(* IEC 61131-3 sources: elnaProjects/ElpcLogic/PomarKc7Changed/build_USO_ecl (part 4) *)

      (*Режим ЭГПА остановлен *)
      EGPA_Stop.top := (algManager.mode = ModeGpa.MODE_STOP);

      (*Автомат ШУ включен *)
      Avt_SHU_vkl.top := IM.SingleSignals.SHU_v_GPA_vkluch.Q;

      (*Все исполнительные механизмы выключены *)
      All_IM_Off.top := (IM.mv.onStatus=_statusDualInput.STATUS_OFF) AND (IM.pns.onStatus=_statusDualInput.STATUS_OFF) AND
                        (IM.nu1.onStatus=_statusDualInput.STATUS_OFF) AND (IM.nu2.onStatus=_statusDualInput.STATUS_OFF) AND
                        (IM.v1_Avom.onStatus=_statusDualInput.STATUS_OFF) AND (IM.v2_Avom.onStatus=_statusDualInput.STATUS_OFF) AND
  		  (IM.v3_Avom.onStatus=_statusDualInput.STATUS_OFF)AND (IM.v4_Avom.onStatus=_statusDualInput.STATUS_OFF) AND
                        (IM.CMN.onStatus=_statusDualInput.STATUS_OFF) AND (IM.TEN_MB.onStatus=_statusDualInput.STATUS_OFF) AND
                        (IM.TEN_kollectora.onStatus=_statusDualInput.STATUS_OFF) AND (IM.KaloriferAVOM.onStatus=_statusDualInput.STATUS_OFF);

      (*Наличие 220 в шу*)
      Nalichie220_SHU_Ai.top :=	(ai.Kontrol_per_220V.interval = _statusAi.normal)	 AND (ai.Kontrol_post_220V.interval = _statusAi.normal);

      (*Блоки питания норм*)
      BP_Norm.top:=
  		(IM.SingleSignals.Nalichie_BP1.Q AND
  		IM.SingleSignals.Nalichie_BP2.Q AND
  		IM.SingleSignals.Nalichie_BP3.Q AND
  		IM.SingleSignals.Nalichie_BP4.Q AND
  		IM.SingleSignals.Nalichie_BP5.Q AND
  		IM.SingleSignals.Nalichie_BP6.Q AND
  		IM.SingleSignals.Nalichie_BP7_BP8.Q AND
  		IM.SingleSignals.Nalichie_BP9_BP10.Q AND

  		IM.SingleSignals.Nalichie_220BEAO.Q AND
  		IM.SingleSignals.Nalichie_per_220_na_vhode.Q AND
  		IM.SingleSignals.Nalichie_post_220_na_vhode.Q AND
  		IM.SingleSignals.Nalichie_BP11.Q AND
  		IM.SingleSignals.Nalichie_BP12.Q);

      (*Напряжение исполнительниых механизмов
      Naprajenie_U_IM.top := IM.NalichieU_CMN.q AND IM.NalichieU_NU1.Q AND IM.Nalichie_CU_MV.Q  AND IM.NalichieU_NU2.Q AND
  						IM.NalichieU_PNS.Q; нет сигналов таких *)

      (* положение тележки мв вкачена *)
      MV_Poloj_RolledON.top:= IM.mv.basketStatus = _basketStats.BASKET_ROLLEDIN;

      (* положение тележки мв выкачена *)
      MV_Poloj_RolledOFF.top:= IM.mv.basketStatus = _basketStats.BASKET_ROLLEDOUT;

      (* нет неисправных аналоговых сигналов *)
      NOTAnalogNS.top :=  NOT analogsNS();

      (* нет аварийных/предупредительных сигнализаций аналоговых сигналов *)
      Net_ASPS_Analogs.top := anyAnalogsPs(); (*Не понял где посмотреть наличие ас аналогов *)

      (* нет сработанных защит *)
      Not_AS.top := NOT anyProtectionSignaling();

      (* готовность возбудителя *)
      Gotov_Vozb.top:= IM.SingleSignals.Vozbud_gotovnost.Q;

      (* реакторный пуск *)
      (*Reactornyi_P.top := IM.SingleSignals.Reaktornii_pusk_perek.Q AND NOT IM.SingleSignals.Chastotny_pusk.Q;*)

      (* частотный пуск *)
     (* Chastotnyi_P.top:=IM.SingleSignals.Chastotny_pusk.Q AND NOT IM.SingleSignals.Reaktornii_pusk_perek.Q;*)

      (* нет перепада давления на кране 1 *)
      dP_kr1.top:= NOT IM.SingleSignals.dp_kran1_Less100.Q (*AND (IM.PerepadDavlenieKran1_CK.status = 1))*);

      (* в автоматическом ли режиме исполнительные механизмы *)
      (*Auto_Rej.top := im.NU1_Automat.Q AND im.PNS_Automat.Q AND im.NU2_Automat.Q;*)

      (* есть наряжение в цепях управления ИМ *)
      CK_IM_Norm.top := nsCepeiUpravlenya();

      (* ручной режим *)
      HAnd_Mode.top:= NOT im.SingleSignals.Rezhim_ruchnogo_regulirovaniya.Q;

      (* импульсный газ *)
      Impuls_Gaz.top:= ai.Pimpuls_gaz.interval=_statusAi.normal;

      ppuDone := BMP_Err.top AND
  	     Level_masla_Norm.top AND
                 T_masla_Norm.top AND
  	     Krans_ready_to_move.top AND
  	     Krans_Poloj.top AND
  	     Net_AO_KC_SHKS04M.top AND
  	     EGPA_Stop.top AND
                 Avt_SHU_vkl.top AND
                 All_IM_Off.top AND
                 Nalichie220_SHU_Ai.top AND
                 BP_Norm.top AND
                 Naprajenie_U_IM.top AND
                 MV_Poloj_RolledON.top AND
                 MV_Poloj_RolledOFF.top AND
                 NOTAnalogNS.top AND
                 Net_ASPS_Analogs.top AND
                 Not_AS.top AND
                 Gotov_Vozb.top AND
                 Reactornyi_P.top AND
                 Chastotnyi_P.top AND
                 dP_kr1.top AND
                 Auto_Rej.top AND
                 CK_IM_Norm.top AND
                 HAnd_Mode.top AND
                 Impuls_Gaz.top;

      puskAllowed:= ppuDone AND Im.mv.basketStatus = _basketStats.BASKET_ROLLEDIN;
      testAllowed:= ppuDone AND Im.mv.basketStatus = _basketStats.BASKET_ROLLEDOUT;

      modeR_Trig(CLK:=puskAllowed);
      modeF_Trig(CLK:=puskAllowed);

      IF modeR_Trig.Q THEN
  	algManager.nMode:= ModeGpa.MODE_READY;
      END_IF;
      IF modeF_Trig.Q THEN
  	algManager.nMode:= ModeGpa.MODE_STOP;
      END_IF;

      IF puskAllowed THEN
          algoritms.Apusk.inCanRun:= TRUE;
          algoritms.SemiAutoPusk.inCanRun:= TRUE;
      ELSE
          algoritms.Apusk.inCanRun:= FALSE;
          algoritms.SemiAutoPusk.inCanRun:= FALSE;
      END_IF;

      IF testAllowed THEN
          algoritms.testPms.inCanRun:=  TRUE;
          algoritms.testdPmg.inCanRun:= TRUE;
          algoritms.puskK.inCanRun:=    TRUE;
          algoritms.puskV.inCanRun:=    TRUE;
      ELSE
          algoritms.testPms.inCanRun:=  FALSE;
          algoritms.testdPmg.inCanRun:= FALSE;
          algoritms.puskK.inCanRun:=    FALSE;
          algoritms.puskV.inCanRun:=    FALSE;
      END_IF;

  END_IF;

  StrAlg.CanRun := StrAlg.inCanRun;
  StrAlg.OpcCommandsDisabled := StrAlg.inOpcCommandsDisabled;

  (* ---- Если управление с ВУ заблокировано, то  передаем команду из алгоритма ---- *)
  IF StrAlg.inOpcCommandsDisabled THEN
  	StrAlg.inCommand := StrAlg.inCommand_Alg;
  ELSE (* иначе передаем команду с АРМа*)
  	StrAlg.inCommand := StrAlg.inCommand_ARM;
  END_IF;

  _sunpackerCommand(command := StrAlg.inCommand);
  	source := _sunpackerCommand.source;
  	cmd := _sunpackerCommand.cmd;

  IF cmd <> 0 AND lastCmd <> cmd AND (((NOT StrAlg.opcCommandsDisabled) AND source > 0) OR source = 0) then
  	CASE BYTE_TO_INT(cmd) OF
  		(*cmdRun*) 1: 	IF (StrAlg.CanRun) THEN
  					StrAlg.isRuning := TRUE;
  					StrAlg.isEnded := FALSE;
  					StrAlg.hasError := FALSE;
  					(*****************       OnRun       *****************)

  					cmd_for_Status := cmd;
  					source_for_Status := source;
  					command_error_for_Status := 0;
  				ELSE
  					StrAlg.isRuning := FALSE;
  					StrAlg.isEnded := FALSE;
  					StrAlg.hasError 	:= FALSE;

  					cmd_for_Status := 0;
  					source_for_Status := source;
  					command_error_for_Status := cmd;
  				END_IF;
  		(*cmdReset*) 2: 	StrAlg.isRuning := FALSE;
  				StrAlg.isEnded := FALSE;
  				StrAlg.hasError 	:= FALSE;

                                           (*****************       OnReset       *****************)

                                                    resetPhase(BMP_Err);
                                                    resetPhase(Level_masla_Norm);
                                                    resetPhase(T_masla_Norm);
                                                    resetPhase(Krans_ready_to_move);
                                                    resetPhase(Krans_Poloj);
                                                    resetPhase(Net_AO_KC_SHKS04M);
                                                    resetPhase(EGPA_Stop);
                                                    resetPhase(Avt_SHU_vkl);
                                                    resetPhase(All_IM_Off);
                                                    resetPhase(Nalichie220_SHU_Ai);
                                                    resetPhase(BP_Norm);
                                                    resetPhase(Naprajenie_U_IM);
                                                    resetPhase(MV_Poloj_RolledON);
                                                    resetPhase(MV_Poloj_RolledOFF);
                                                    resetPhase(NOTAnalogNS);
                                                    resetPhase(Net_ASPS_Analogs);
                                                    resetPhase(Not_AS);
                                                    resetPhase(Gotov_Vozb);
                                                    resetPhase(Reactornyi_P);
                                                    resetPhase(Chastotnyi_P);
                                                    resetPhase(dP_kr1);
                                                    resetPhase(Auto_Rej);
                                                    resetPhase(CK_IM_Norm);
                                                    resetPhase(HAnd_Mode);
                                                    resetPhase(Impuls_Gaz);

                                                    algoritms.testPms.inCanRun:=  FALSE;
                                                    algoritms.testdPmg.inCanRun:= FALSE;
                                                    algoritms.puskK.inCanRun:=    FALSE;
                                                    algoritms.puskV.inCanRun:=    FALSE;

                                          StrAlg.inCanRun:=FALSE;
                                          puskAllowed:=FALSE;
                                          testAllowed:=FALSE;
                                          modeR_Trig(CLK:=FALSE);
                                          modeF_Trig(CLK:=FALSE);

  				cmd_for_Status := cmd;
  				source_for_Status := source;
  				command_error_for_Status := 0;
  	END_CASE;
  	resetCmdTimer(IN := false);
  	resetCmdTimerPriznak := TRUE;
  END_IF;
  lastCmd := cmd;

  resetCmdTimer(IN := resetCmdTimerPriznak, PT := T#5S);
  IF resetCmdTimer.Q THEN
  	resetCmdTimerPriznak := FALSE;
  	source_for_Status := 0;
  	cmd_for_Status := 0;
  	command_error_for_Status := 0;
  END_IF;

  StrAlg.Start:= BMP_Err.startStatus
              OR Level_masla_Norm.startStatus
              OR T_masla_Norm.startStatus
              OR Krans_ready_to_move.startStatus
              OR Krans_Poloj.startStatus
              OR Net_AO_KC_SHKS04M.startStatus
              OR EGPA_Stop.startStatus
              OR Avt_SHU_vkl.startStatus
              OR All_IM_Off.startStatus
              OR Nalichie220_SHU_Ai.startStatus
              OR BP_Norm.startStatus
              OR Naprajenie_U_IM.startStatus
              OR MV_Poloj_RolledON.startStatus
              OR MV_Poloj_RolledOFF.startStatus
              OR NOTAnalogNS.startStatus
              OR Net_ASPS_Analogs.startStatus
              OR Not_AS.startStatus
              OR Gotov_Vozb.startStatus
              OR Reactornyi_P.startStatus
              OR Chastotnyi_P.startStatus
              OR dP_kr1.startStatus
              OR Auto_Rej.startStatus
              OR CK_IM_Norm.startStatus
              OR HAnd_Mode.startStatus
              OR Impuls_Gaz.startStatus;

  StrAlg.Error:= BMP_Err.errorStatus
              OR Level_masla_Norm.errorStatus
              OR T_masla_Norm.errorStatus
              OR Krans_ready_to_move.errorStatus
              OR Krans_Poloj.errorStatus
              OR Net_AO_KC_SHKS04M.errorStatus
              OR EGPA_Stop.errorStatus
              OR Avt_SHU_vkl.errorStatus
              OR All_IM_Off.errorStatus
              OR Nalichie220_SHU_Ai.errorStatus
              OR BP_Norm.errorStatus
              OR Naprajenie_U_IM.errorStatus
              OR MV_Poloj_RolledON.errorStatus
              OR MV_Poloj_RolledOFF.errorStatus
              OR NOTAnalogNS.errorStatus
              OR Net_ASPS_Analogs.errorStatus
              OR Not_AS.errorStatus
              OR Gotov_Vozb.errorStatus
              OR Reactornyi_P.errorStatus
              OR Chastotnyi_P.errorStatus
              OR dP_kr1.errorStatus
              OR Auto_Rej.errorStatus
              OR CK_IM_Norm.errorStatus
              OR HAnd_Mode.errorStatus
              OR Impuls_Gaz.errorStatus;

  StrAlg.Top:=   BMP_Err.topStatus
              OR Level_masla_Norm.topStatus
              OR T_masla_Norm.topStatus
              OR Krans_ready_to_move.topStatus
              OR Krans_Poloj.topStatus
              OR Net_AO_KC_SHKS04M.topStatus
              OR EGPA_Stop.topStatus
              OR Avt_SHU_vkl.topStatus
              OR All_IM_Off.topStatus
              OR Nalichie220_SHU_Ai.topStatus
              OR BP_Norm.topStatus
              OR Naprajenie_U_IM.topStatus
              OR MV_Poloj_RolledON.topStatus
              OR MV_Poloj_RolledOFF.topStatus
              OR NOTAnalogNS.topStatus
              OR Net_ASPS_Analogs.topStatus
              OR Not_AS.topStatus
              OR Gotov_Vozb.topStatus
              OR Reactornyi_P.topStatus
              OR Chastotnyi_P.topStatus
              OR dP_kr1.topStatus
              OR Auto_Rej.topStatus
              OR CK_IM_Norm.topStatus
              OR HAnd_Mode.topStatus
              OR Impuls_Gaz.topStatus;

  (*TODO: TYPE PROGRAM CODE HERE*)
  StrAlg.status :=  SHL(BYTE_TO_DWORD(source_for_Status), 29)
  			OR SHL(BYTE_TO_DWORD(cmd_for_Status), 26)
  			OR SHL(BYTE_TO_DWORD(command_error_for_Status), 23)
  			OR SHL(BOOL_TO_DWORD(StrAlg.OpcCommandsDisabled ), 21)
                                OR SHL(BOOL_TO_DWORD(testAllowed),16)
                                OR SHL(BOOL_TO_DWORD(puskAllowed),15)
  			OR SHL(BOOL_TO_DWORD(StrAlg.hasError),4)
  			OR SHL(BOOL_TO_DWORD(StrAlg.CanRun),2)
  			OR SHL(BOOL_TO_DWORD(StrAlg.isEnded),1)
  			OR BOOL_TO_DWORD(StrAlg.isRuning);
END_FUNCTION_BLOCK

FUNCTION_BLOCK ph_SingleSignal
  VAR_IN_OUT
    im : struct_singleSignal;
  END_VAR
  VAR_INPUT
    expectedValue : BOOL          := TRUE;
    PhaseNumber : UINT;
  END_VAR
  VAR_IN_OUT
    StrPh : struct_PhaseAlgoritm;
  END_VAR
  VAR
    reset_Trig : R_TRIG;
  END_VAR

  IF StrPh.run AND NOT StrPh.start THEN
  	StrPh.start := TRUE;
  	StrPh.top := FALSE;
  	StrPh.error := FALSE;
            StrPh.run:=FALSE;
  END_IF;

  IF StrPh.start AND NOT StrPh.top THEN
  StrPh.error:= NOT Im.reliability;
  StrPh.top := (Im.Q = expectedValue) AND (Im.reliability);
  END_IF;

  reset_Trig(CLK := StrPh.reset);
  IF reset_Trig.Q THEN
  	StrPh.start := FALSE;
  	StrPh.error := FALSE;
  	StrPh.top := FALSE;
            StrPh.run:=FALSE;
            StrPh.reset:=FALSE;
  END_IF;

  StrPh.startStatus := SHL(BOOL_TO_DWORD(StrPh.start), PhaseNumber);
  StrPh.errorStatus := SHL(BOOL_TO_DWORD(StrPh.error), PhaseNumber);
  StrPh.topStatus := SHL(BOOL_TO_DWORD(StrPh.top), PhaseNumber);
END_FUNCTION_BLOCK

FUNCTION_BLOCK fb_ph_WaitAnalogValue
  VAR_IN_OUT
    ai : struct_AI;
  END_VAR
  VAR_INPUT
    more : LREAL;
    less : LREAL;
    PhaseNumber : UINT;
  END_VAR
  VAR_IN_OUT
    StrPh : struct_PhaseAlgoritm;
  END_VAR
  VAR
    CommandFault_Trig : R_TRIG;
    reset_Trig : R_TRIG;
    _statusAi : TYPE_StatusAi;
    _statusDualInput : TYPE_statusDualInput;
  END_VAR

  IF StrPh.run AND NOT StrPh.start THEN
  	StrPh.start := TRUE;
  	StrPh.top := FALSE;
  	StrPh.error := FALSE;
            StrPh.run:=FALSE;
  END_IF;

  IF StrPh.start AND NOT StrPh.top THEN
                      IF ai.interval < _statusAi.normal THEN
  	              StrPh.error := TRUE;
                          StrPh.top:=FALSE;
                      ELSE
                              IF (more<>0.0) OR (less<>0.0) THEN
                              StrPh.top:=TRUE;
  	                    IF more<>0.0 THEN StrPh.top:=StrPh.top AND (ai.value > more); END_IF;
  	                    IF less<>0.0 THEN StrPh.top:=StrPh.top AND (ai.value < less); END_IF;
                              ELSE
  	                  StrPh.top:=TRUE;
                              END_IF;
                     END_IF;
  END_IF;

  IF StrPh.top THEN
  StrPh.error := FALSE;
  END_IF;

  reset_Trig(CLK := StrPh.reset);
  IF reset_Trig.Q THEN
  	StrPh.start := FALSE;
  	StrPh.error := FALSE;
  	StrPh.top := FALSE;
            StrPh.run:=FALSE;
            StrPh.reset:=FALSE;
  END_IF;

  StrPh.startStatus := SHL(BOOL_TO_DWORD(StrPh.start), PhaseNumber);
  StrPh.errorStatus := SHL(BOOL_TO_DWORD(StrPh.error), PhaseNumber);
  StrPh.topStatus := SHL(BOOL_TO_DWORD(StrPh.top), PhaseNumber);
END_FUNCTION_BLOCK

FUNCTION_BLOCK fb_TableValue_Min
  VAR_INPUT
    parametr : REAL;
  END_VAR
  VAR
    _table : ARRAY [0..8] OF TYPE_TableRec;
  END_VAR
  VAR_INPUT
    inverse : BOOL          := FALSE;
  END_VAR
  VAR_IN_OUT
    actualValue : REAL;
  END_VAR
  VAR
    indexLess : INT          := -1;
    indexMore : INT          := -1;
    Vali : REAL;
    i : INT;
    moreDistance : REAL;
    lessDistance : REAL;
    onInit : BOOL;
    _prevParam : REAL          := 50.0;
  END_VAR
  VAR CONSTANT
    maxTableLength : INT          := 9;
  END_VAR

  IF NOT onInit THEN
  _table[0].x:=-35.0;  _table[0].y:=130.0;
  _table[1].x:=-25.0;  _table[1].y:=124.0;
  _table[2].x:=-15.0;  _table[2].y:=118.0;
  _table[3].x:= -5.0;  _table[3].y:=112.0;
  _table[4].x:=  0.0;  _table[4].y:=108.0;
  _table[5].x:=  5.0;  _table[5].y:=106.0;
  _table[6].x:= 15.0;  _table[6].y:=104.0;
  _table[7].x:= 25.0;  _table[7].y:=102.0;
  _table[8].x:= 35.0;  _table[8].y:= 97.0;

  onInit:=TRUE;
  END_IF;

  IF parametr <> _prevParam THEN
  indexLess:=-1;
  indexMore:=-1;
  lessDistance:=0.0;
  moreDistance:=0.0;
  FOR i:=0 TO maxTableLength-1 DO
  	IF NOT inverse THEN
  		Vali:=_table[i].x;
  	ELSE
  		Vali:=_table[i].y;
  	END_IF;

  	IF (Vali=parametr) THEN
  		indexLess:=i;
  		indexMore:=i;
  	ELSIF ((Vali<parametr) AND ((lessDistance>parametr-Vali) OR (indexLess<0))) THEN
  		indexLess:=i;
  		lessDistance:=parametr-Vali;
  	ELSIF ((Vali>parametr) AND ((moreDistance>Vali-parametr) OR (indexMore<0))) THEN
  		indexMore:=i;
  		moreDistance:=parametr-Vali;
  	END_IF;
  END_FOR;
  (*
  IF indexLess<0 THEN
  	indexLess:=indexMore;
  END_IF;

  IF indexMore<0 THEN
  	indexMore:=indexLess;
  END_IF;
  *)
    IF (_table[indexMore].x<>_table[indexLess].x) THEN
    actualValue:=_table[indexLess].y+((_table[indexMore].y-_table[indexLess].y)/(_table[indexMore].x-_table[indexLess].x))*(parametr-_table[indexLess].x);
    ELSE
    actualValue:=_table[indexLess].y;
    END_IF;
     _prevParam:= parametr;
  END_IF;
END_FUNCTION_BLOCK

FUNCTION_BLOCK fb_TableValue_Max
  VAR_INPUT
    parametr : REAL;
  END_VAR
  VAR
    _table : ARRAY [0..8] OF TYPE_TableRec;
  END_VAR
  VAR_INPUT
    inverse : BOOL          := FALSE;
  END_VAR
  VAR_IN_OUT
    actualValue : REAL;
  END_VAR
  VAR
    indexLess : INT          := -1;
    indexMore : INT          := -1;
    Vali : REAL;
    i : INT;
    moreDistance : REAL;
    lessDistance : REAL;
    onInit : BOOL;
    _prevParam : REAL          := 50.0;
  END_VAR
  VAR CONSTANT
    maxTableLength : INT          := 9;
  END_VAR

  IF NOT onInit THEN
  _table[0].x:=-35.0;  _table[0].y:=320.0;
  _table[1].x:=-25.0;  _table[1].y:=315.0;
  _table[2].x:=-15.0;  _table[2].y:=310.0;
  _table[3].x:= -5.0;  _table[3].y:=305.0;
  _table[4].x:=  0.0;  _table[4].y:=300.0;
  _table[5].x:=  5.0;  _table[5].y:=295.0;
  _table[6].x:= 15.0;  _table[6].y:=290.0;
  _table[7].x:= 25.0;  _table[7].y:=285.0;
  _table[8].x:= 35.0;  _table[8].y:=280.0;

  onInit:=TRUE;
  END_IF;

  IF parametr <> _prevParam THEN
  indexLess:=-1;
  indexMore:=-1;
  lessDistance:=0.0;
  moreDistance:=0.0;
  FOR i:=0 TO maxTableLength-1 DO
  	IF NOT inverse THEN
  		Vali:=_table[i].x;
  	ELSE
  		Vali:=_table[i].y;
  	END_IF;

  	IF (Vali=parametr) THEN
  		indexLess:=i;
  		indexMore:=i;
  	ELSIF ((Vali<parametr) AND ((lessDistance>parametr-Vali) OR (indexLess<0))) THEN
  		indexLess:=i;
  		lessDistance:=parametr-Vali;
  	ELSIF ((Vali>parametr) AND ((moreDistance>Vali-parametr) OR (indexMore<0))) THEN
  		indexMore:=i;
  		moreDistance:=parametr-Vali;
  	END_IF;
  END_FOR;
  (*
  IF indexLess<0 THEN
  	indexLess:=indexMore;
  END_IF;

  IF indexMore<0 THEN
  	indexMore:=indexLess;
  END_IF;
  *)
    IF (_table[indexMore].x<>_table[indexLess].x) THEN
    actualValue:=_table[indexLess].y+((_table[indexMore].y-_table[indexLess].y)/(_table[indexMore].x-_table[indexLess].x))*(parametr-_table[indexLess].x);
    ELSE
    actualValue:=_table[indexLess].y;
    END_IF;
     _prevParam:= parametr;
  END_IF;
END_FUNCTION_BLOCK

FUNCTION_BLOCK fb_ZapasAlg
  VAR_INPUT
    Q_actual : struct_AI;
  END_VAR
  VAR_IN_OUT
    StrAi : struct_AI;
  END_VAR
  VAR_INPUT
    Q_min : LREAL;
    Q_max : LREAL;
  END_VAR
  VAR
    _statusAi : TYPE_StatusAi;
  END_VAR

  IF (Q_actual.interval < _statusAi.normal) THEN
  	StrAi.interval := _statusAi.NOTRELIABLE;
            strAI.status := 	SHL(BOOL_TO_DWORD(strAI.OpcCommandsDisabled ), 21)
  		OR BYTE_TO_DWORD(strAI.interval);
  	RETURN;
  END_IF;

  IF (Q_actual.value <10.0) THEN
  	StrAi.interval := _statusAi.normal;
  	StrAi.value:= 100.0;
            strAI.status := 	SHL(BOOL_TO_DWORD(strAI.OpcCommandsDisabled ), 21)
  		OR BYTE_TO_DWORD(strAI.interval);
  	RETURN;
  END_IF;

  strAI.opcCommandsDisabled := strAI.inopcCommandsDisabled ;
  StrAi.interval:= _statusAi.normal;

  StrAi.value:= ((Q_actual.value - Q_min)/(Q_max-Q_min))*100.0;

  strAI.status := 	SHL(BOOL_TO_DWORD(strAI.OpcCommandsDisabled ), 21) (* Управление в ВУ заблокировано *)
  		OR BYTE_TO_DWORD(strAI.interval);	              (* интервал *)
END_FUNCTION_BLOCK

FUNCTION_BLOCK fb_AntiPompagAlg
  VAR
    tableQ_min : fb_TableValue_Min;
    tableQ_max : fb_TableValue_Max;
    fb_Rashod : fb_RashodAlg;
    fb_Zapas : fb_ZapasAlg;
  END_VAR
  VAR_IN_OUT
    Kran6 : struct_Kran;
    StrAlg : struct_Alg;
    Rashod : struct_AI;
    Zapas : struct_AI;
  END_VAR
  VAR_INPUT
    P_gasIn : struct_AI;
    T_gasIn : struct_AI;
    dP_konf : struct_AI;
    UgolVNA : struct_AnalogParametr;
    K : struct_AnalogParametr;
    A : struct_AnalogParametr;
    y0 : struct_AnalogParametr;
  END_VAR
  VAR
    Q_max : LREAL;
    Q_min : LREAL;
    pompaj : BOOL;
    _statusAi : TYPE_StatusAi;
    _statusDualInput : TYPE_statusDualInput;
    _sunpackerCommand : fb_sunpackerCommand;
    source : BYTE;
    cmd : BYTE;
    lastCmd : BYTE;
    source_for_Status : BYTE;
    cmd_for_Status : BYTE;
    command_error_for_Status : BYTE;
    resetCmdTimer : TON;
    resetCmdTimerPriznak : BOOL;
  END_VAR

  tableQ_min(parametr:=LREAL_TO_REAL(UgolVNA.Value));

  tableQ_max(parametr:=LREAL_TO_REAL(UgolVNA.Value));

  Q_min:=REAL_TO_LREAL(tableQ_min.actualValue);

  Q_max:=REAL_TO_LREAL(tableQ_max.actualValue);

  fb_Rashod(StrAi:=Rashod, P_gasIn:=P_gasIn, T_gasIn:=T_gasIn, dP_konf:=dP_konf, K:=K, A:=A, y0:=y0);

  fb_Zapas(StrAi:=Zapas, Q_actual:=Rashod, Q_min:=Q_min, Q_max:=Q_max);

  StrAlg.CanRun := StrAlg.inCanRun;

  StrAlg.OpcCommandsDisabled := StrAlg.inOpcCommandsDisabled;

  IF StrAlg.isRuning THEN

  StrAlg.hasError := (Rashod.interval < _statusAi.normal);

  pompaj:= (Rashod.interval>=_statusAi.normal) AND (Rashod.value <= Q_min);

  IF pompaj THEN
            Kran6.inOpcCommandsDisabled:=TRUE;
  	Kran6.inCommand_Alg := 1;  (*cmd_open*)
  END_IF;

  StrAlg.isEnded := Kran6.onStatus = _statusDualInput.STATUS_ON ;

  END_IF;

  (* ---- Если управление с ВУ заблокировано, то передаем команду из алгоритма ---- *)
  IF StrAlg.inOpcCommandsDisabled THEN
  	StrAlg.inCommand := StrAlg.inCommand_Alg;
  ELSE (* иначе передаем команду с АРМа*)
  	StrAlg.inCommand := StrAlg.inCommand_ARM;
  END_IF;

  _sunpackerCommand(command := StrAlg.inCommand);
  	source := _sunpackerCommand.source;
  	cmd := _sunpackerCommand.cmd;

  IF cmd <> 0 AND lastCmd <> cmd AND (((NOT StrAlg.opcCommandsDisabled) AND source > 0) OR source = 0) then
  	CASE BYTE_TO_INT(cmd) OF
  		(*cmdRun*) 1: 	IF (StrAlg.CanRun) THEN
  					StrAlg.isRuning := TRUE;
  					StrAlg.isEnded := FALSE;
  					StrAlg.hasError 	:= FALSE;

                                                    (*****************       OnRun       *****************)

  					cmd_for_Status := cmd;
  					source_for_Status := source;
  					command_error_for_Status := 0;
  				ELSE
  					StrAlg.isRuning := FALSE;
  					StrAlg.isEnded := FALSE;
  					StrAlg.hasError 	:= FALSE;

  					cmd_for_Status := 0;
  					source_for_Status := source;
  					command_error_for_Status := cmd;
  				END_IF;
  		(*cmdReset*) 2: 	StrAlg.isRuning := FALSE;
  				StrAlg.isEnded := FALSE;
  				StrAlg.hasError 	:= FALSE;
                                          (*****************       OnReset       *****************)

                                                    pompaj:= FALSE;
                                                    Kran6.inOpcCommandsDisabled:=FALSE;
  				cmd_for_Status := cmd;
  				source_for_Status := source;
  				command_error_for_Status := 0;
  	END_CASE;
  	resetCmdTimer(IN := false);
  	resetCmdTimerPriznak := TRUE;
  END_IF;
  lastCmd := cmd;

  resetCmdTimer(IN := resetCmdTimerPriznak, PT := T#5S);
  IF resetCmdTimer.Q THEN
  	resetCmdTimerPriznak := FALSE;
  	source_for_Status := 0;
  	cmd_for_Status := 0;
  	command_error_for_Status := 0;
  END_IF;

  StrAlg.status :=  SHL(BYTE_TO_DWORD(source_for_Status), 29)
  			OR SHL(BYTE_TO_DWORD(cmd_for_Status), 26)
  			OR SHL(BYTE_TO_DWORD(command_error_for_Status), 23)
  			OR SHL(BOOL_TO_DWORD(StrAlg.OpcCommandsDisabled ), 21)
  			OR SHL(BOOL_TO_DWORD(StrAlg.hasError),4)
  			OR SHL(BOOL_TO_DWORD(StrAlg.CanRun),2)
  			OR SHL(BOOL_TO_DWORD(StrAlg.isEnded),1)
  			OR BOOL_TO_DWORD(StrAlg.isRuning);
END_FUNCTION_BLOCK

FUNCTION_BLOCK fb_AnalogParametr_Init
  VAR_INPUT
    data_Ini : BOOL;
    currentValue : LREAL;
    minVal : LREAL;
    maxVal : LREAL;
    maxStep : LREAL;
    minVal_ISVALIDREF : BOOL;
    maxVal_ISVALIDREF : BOOL;
    maxStep_ISVALIDREF : BOOL;
  END_VAR
  VAR_IN_OUT
    strAP : struct_AnalogParametr;
  END_VAR
  VAR_OUTPUT
    Init : BOOL          := FALSE;
  END_VAR

  (*****            Функциональный блок переинициализации Аналогового параметра.            *****)
       Init := false;

      IF data_Ini THEN                            (* Параметрам требуется переинициализация. *)
          strAP.currentValue          := currentValue;
          strAP.minVal                := minVal;
          strAP.maxVal                := maxVal;
          strAP.maxStep               := maxStep;
          strAP.minVal_ISVALIDREF     := minVal_ISVALIDREF;
          strAP.maxVal_ISVALIDREF     := maxVal_ISVALIDREF;
          strAP.maxStep_ISVALIDREF    := maxStep_ISVALIDREF;

          data_Ini:=false;
          Init := TRUE;
       END_IF;
       IF Init THEN
          currentValue:= 0.0;
          minVal:= 0.0;
          maxVal:= 0.0;
          maxStep:= 0.0;
          minVal_ISVALIDREF:= false;
          maxVal_ISVALIDREF:= false;
          maxStep_ISVALIDREF:= false;
       END_IF;
END_FUNCTION_BLOCK

FUNCTION_BLOCK proc_DO
  VAR
    do_0 : fb_DOSourceMlp;
    do_1 : fb_DOSourceMlp;
    do_2 : fb_DOSourceMlp;
    do_3 : fb_DOSourceMlp;
    do_4 : fb_DOSourceMlp;
    gpio_out : fb_DOSourceMlp;
  END_VAR
  VAR_EXTERNAL
    od : DOconfig;
    arDOUT_0 : TWordData;
    arDOUT_1 : TWordData;
    arDOUT_2 : TWordData;
    arDOUT_3 : TWordData;
    arDOUT_4 : TWordData;
    arERR_66 : TItemDIN;
    arDOUT_66 : TWordData;
    arERR_0 : TItemDIN;
    arERR_1 : TItemDIN;
    arERR_2 : TItemDIN;
    arERR_15 : TItemDIN;
    arERR_16 : TItemDIN;
    A1_1_err_mode : UINT;
    A1_2_err_mode : UINT;
    A1_3_err_mode : UINT;
    A2_1_err_mode : UINT;
    A2_4_err_mode : UINT;
    DO_0_wValue : UINT;
    DO_1_wValue : UINT;
    DO_2_wValue : UINT;
    DO_3_wValue : UINT;
    DO_4_wValue : UINT;
  END_VAR

  (* Циклический опрос. Входные дискретные параметры *)

  (* Модуль A1-1 *)
  do_0(arDout := arDOUT_0, strDO := od.do_0, err_mod:=arERR_0);
  DO_0_wValue:=arDOUT_0.wValue;
  A1_1_err_mode:= arERR_0.wValue;

  (* Модуль A1-2 *)
  do_1(arDout := arDOUT_1, strDO := od.do_1, err_mod:=arERR_1);
  DO_1_wValue:=arDOUT_1.wValue;
  A1_2_err_mode:= arERR_1.wValue;

  (* Модуль A1-3 *)
  do_2(arDout := arDOUT_2, strDO := od.do_2, err_mod:=arERR_2);
  DO_2_wValue:=arDOUT_2.wValue;
  A1_3_err_mode:= arERR_2.wValue;

  (* Модуль A2-1 *)
  do_3(arDout := arDOUT_3, strDO := od.do_3, err_mod:=arERR_15);
  DO_3_wValue:=arDOUT_3.wValue;
  A2_1_err_mode:= arERR_15.wValue;

  (* Модуль A2-1 *)
  do_4(arDout := arDOUT_4, strDO := od.do_4, err_mod:=arERR_15);
  DO_4_wValue:=arDOUT_4.wValue;
  A2_4_err_mode:= arERR_16.wValue;

  gpio_out(arDout := arDOUT_66, strDO := od.gpio_out, err_mod:=arERR_66);
END_FUNCTION_BLOCK

FUNCTION_BLOCK proc_DI_Init
  VAR_INPUT
    init : BOOL;
  END_VAR
  VAR
    stDI_Ini : fb_DI_Init;
    inits : UINT;
  END_VAR
  VAR_INPUT
    initiales : UINT;
  END_VAR
  VAR_EXTERNAL
    di : DiConfig;
  END_VAR

  (* Инициализация начало. Входные дискретные параметры *)

  inits := 0; (* Флаг необходимости инициализации структур-дескрипторов *)

  (* Модуль A1-1 *)

  stDI_Ini(data_Ini := true, imit:=FALSE, strDI := di.di_0);
  inits := inits + BOOL_TO_UINT(stDI_Ini.Init);

  stDI_Ini(data_Ini := true, imit:=FALSE, strDI := di.di_1);
  inits := inits + BOOL_TO_UINT(stDI_Ini.Init);

  (* Модуль A1-2 *)
  stDI_Ini(data_Ini := true, imit:=FALSE, strDI := di.di_2);
  inits := inits + BOOL_TO_UINT(stDI_Ini.Init);

  stDI_Ini(data_Ini := true, imit:=FALSE, strDI := di.di_3);
  inits := inits + BOOL_TO_UINT(stDI_Ini.Init);

  (* Модуль A1-3 *)
  stDI_Ini(data_Ini := true, imit:=FALSE, strDI := di.di_4);
  inits := inits + BOOL_TO_UINT(stDI_Ini.Init);

  stDI_Ini(data_Ini := true, imit:=FALSE, strDI := di.di_5);
  inits := inits + BOOL_TO_UINT(stDI_Ini.Init);

  (* Модуль A1-4 *)
  stDI_Ini(data_Ini := true, imit:=FALSE, strDI := di.di_6);
  inits := inits + BOOL_TO_UINT(stDI_Ini.Init);

  stDI_Ini(data_Ini := true, imit:=FALSE, strDI := di.di_7);
  inits := inits + BOOL_TO_UINT(stDI_Ini.Init);

  (* Модуль A1-5 *)
  stDI_Ini(data_Ini := true, imit:=FALSE,  strDI := di.di_8);
  inits := inits + BOOL_TO_UINT(stDI_Ini.Init);

  stDI_Ini(data_Ini := true, imit:=FALSE,  strDI := di.di_9);
  inits := inits + BOOL_TO_UINT(stDI_Ini.Init);

  (* Модуль A1-6 *)
  stDI_Ini(data_Ini := true, imit:=FALSE,  strDI := di.di_10);
  inits := inits + BOOL_TO_UINT(stDI_Ini.Init);

  stDI_Ini(data_Ini := true, imit:=FALSE,  strDI := di.di_11);
  inits := inits + BOOL_TO_UINT(stDI_Ini.Init);

  (* Модуль A1-7 *)
  stDI_Ini(data_Ini := true, imit:=FALSE, strDI := di.di_12);
  inits := inits + BOOL_TO_UINT(stDI_Ini.Init);

  stDI_Ini(data_Ini := true, imit:=FALSE, strDI := di.di_13);
  inits := inits + BOOL_TO_UINT(stDI_Ini.Init);

  (* Модуль A1-8 *)
  stDI_Ini(data_Ini := true, imit:=FALSE, strDI := di.di_14);
  inits := inits + BOOL_TO_UINT(stDI_Ini.Init);

  stDI_Ini(data_Ini := true, imit:=FALSE, strDI := di.di_16);
  inits := inits + BOOL_TO_UINT(stDI_Ini.Init);

  stDI_Ini(data_Ini := true, imit:=FALSE, strDI := di.di_17);
  inits := inits + BOOL_TO_UINT(stDI_Ini.Init);

  stDI_Ini(data_Ini := true, imit:=FALSE, strDI := di.di_18);
  inits := inits + BOOL_TO_UINT(stDI_Ini.Init);

  stDI_Ini(data_Ini := true, imit:=FALSE, strDI := di.di_19);
  inits := inits + BOOL_TO_UINT(stDI_Ini.Init);

  stDI_Ini(data_Ini := true, imit:=FALSE, strDI := di.di_20);
  inits := inits + BOOL_TO_UINT(stDI_Ini.Init);

  stDI_Ini(data_Ini := true, imit:=FALSE, strDI := di.di_21);
  inits := inits + BOOL_TO_UINT(stDI_Ini.Init);

  initiales := 0;
  IF init THEN initiales := inits; END_IF;
END_FUNCTION_BLOCK

FUNCTION_BLOCK fb_Kran
  VAR_INPUT
    statOn : BOOL;
    statOff : BOOL;
    statOn_reliability : BOOL;
    statOff_reliability : BOOL;
  END_VAR
  VAR_IN_OUT
    strKr : struct_Kran;
  END_VAR
  VAR_INPUT
    inNs : TYPE_ReliableBit;
    inAccident : TYPE_ReliableBit;
    inAuto : TYPE_ReliableBit;
    inManual : TYPE_ReliableBit;
    inLocal : TYPE_ReliableBit;
    inDistance : TYPE_ReliableBit;
    inErrorPowerOff : TYPE_ReliableBit;
    inErrorBlock : TYPE_ReliableBit;
    inSo : TYPE_ReliableBit;
    inSz : TYPE_ReliableBit;
    inDp : TYPE_ReliableBit;
  END_VAR
  VAR
    onInit : BOOL          := FALSE;
    _statOn : BOOL;
    _statOff : BOOL;
    getSdvig : BOOL;
    lastOnStatus : BYTE;
    cmd : BYTE;
    source : BYTE;
    lastCmd : BYTE;
    source_for_Status : BYTE;
    cmd_for_Status : BYTE;
    command_error_for_Status : BYTE;
    _sunpackerCommand : fb_sunpackerCommand;
    _statusDualInput : TYPE_statusDualInput;
    _commandDualInput : TYPE_commandDualInput;
    _commandErrorTimer : BOOL;
    resetErrorTimer : BOOL;
    _changWithoutCommand : BOOL;
    BlockedOpenControl : BOOL;
    errorCMDTimer : TON;
    _errorReset : TON;
    sdvigReset : TON;
    continueHoldCommandTimer : TON;
    outputsSets : TOF;
    dP_Trig : R_TRIG;
    dP_Trig_reliability : R_TRIG;
    resetBlockedOpenControl_Trig : R_TRIG;
  END_VAR
  VAR_IN_OUT
    cmdOn : BOOL;
    cmdOff : BOOL;
  END_VAR

  IF NOT onInit THEN
  IF strKr.ISVALIDREF_cmdOn XOR strKr.ISVALIDREF_cmdOff THEN
  	IF 	strKr.ISVALIDREF_cmdOn THEN
  		lastCmd:= 2; (*baseCmdOff*)
  	ELSE
  		lastCmd:= 1; (*baseCmdOn*)
  	END_IF;
  END_IF;
  onInit:=TRUE;
  END_IF;

  (* ---- Если управление с ВУ заблокировано, то в ИМ передаем команду из алгоритма ---- *)
  IF strKr.inOpcCommandsDisabled THEN
  	strKr.inCommand := strKr.inCommand_Alg;
  ELSE (* иначе передаем команду с АРМа*)
  	strKr.inCommand := strKr.inCommand_ARM;
  END_IF;

  (* ---- Формирование состояния механизма ---- *)

  IF (strKr.ISVALIDREF_statOn) OR (strKr.ISVALIDREF_statOff) THEN
  	IF (strKr.ISVALIDREF_statOn) AND (strKr.ISVALIDREF_statOff) THEN
  	strKr.reliability:= statOn_reliability AND statOff_reliability;
  		_statOn  := statOn;
  		_statOff := statOff;
  	ELSIF (strKr.ISVALIDREF_statOn) THEN
                       strKr.reliability:= statOn_reliability;
  		_statOn  := statOn;
  		_statOff := NOT statOn;
  	ELSIF (strKr.ISVALIDREF_statOff) THEN
  		 strKr.reliability:= statOff_reliability;
  		_statOn  := NOT statOff;
  		_statOff :=statOff;
  	END_IF;

  	IF strKr.reliability THEN
  		IF _statOn AND NOT _statOff 		THEN 	strKr.onStatus := _statusDualInput.STATUS_ON;
  		ELSIF _statOff AND NOT _statOn 	THEN 	strKr.onStatus := _statusDualInput.Status_OFF;
  		ELSIF NOT _statOn AND NOT _statOff 	THEN 	strKr.onStatus := _statusDualInput.STATUS_TRANSITIONAL;
  		ELSE					strKr.onStatus := _statusDualInput.STATUS_ERROR;
                      END_IF;

  	ELSE
  		strKr.onStatus := _statusDualInput.STATUS_NOTDEFINED;

  	END_IF;
  ELSE
  	CASE BYTE_TO_INT(lastCmd) OF
  		(*baseCmdOn*)  1: strKr.onStatus  := _statusDualInput.STATUS_ON;
  		(*baseCmdOff*) 2: strKr.onStatus  := _statusDualInput.STATUS_OFF;

  	ELSE
  		 strKr.onStatus := _statusDualInput.STATUS_NOTDEFINED;

  	END_CASE;
  END_IF;

  strKr.Accident := inAccident.value AND inAccident.reliability;
  strKr.Ns := inNs.value AND inNs.reliability;
  strKr.Auto := inAuto.value AND inAuto.reliability;
  strKr.Manual := inManual.value AND inManual.reliability;
  strKr.Local := inLocal.value AND inLocal.reliability;
  strKr.Distance := inDistance.value AND inDistance.reliability;
  strKr.ErrorPowerOff := inErrorPowerOff.value AND inErrorPowerOff.reliability;
  strKr.ErrorBlock := inErrorBlock.value AND inErrorBlock.reliability;
  strKr.OpcCommandsDisabled := strKr.inOpcCommandsDisabled;

  (* ---- Формирование признака блокировки Открытия крана по высокому давлению ---- *)
  	IF strKr.ISVALIDREF_inDp THEN

  		strKr.Dp := NOT inDp.value AND inDp.reliability;

  		dP_Trig(CLK := strKr.Dp );
  		dP_Trig_reliability(CLK :=NOT inDp.reliability);

  		IF dP_Trig.Q OR dP_Trig_reliability.Q THEN
  			BlockedOpenControl := TRUE;
  		END_IF;
  		(* ---- автоматический сброс *)
  		resetBlockedOpenControl_Trig(CLK := (inDp.value) AND inDp.reliability);
  		IF resetBlockedOpenControl_Trig.Q THEN
  			BlockedOpenControl := FALSE;
  		END_IF;
  	ELSE
  		strKr.Dp  := FALSE;
  		BlockedOpenControl := FALSE;
  	END_IF;

  (* ---- Формирование признака сдвига ---- *)
  getSdvig := FALSE;
  IF (strKr.ISVALIDREF_cmdOn OR strKr.ISVALIDREF_cmdOff) AND NOT strKr.Local THEN
  	IF NOT (strKr.CmdOn OR strKr.CmdOff) THEN
  		IF (lastOnStatus <> strKr.onStatus AND
  		(strKr.onStatus <> _statusDualInput.STATUS_NOTDEFINED AND strKr.onStatus <> _statusDualInput.STATUS_ERROR) AND
  		(lastOnStatus <> _statusDualInput.STATUS_NOTDEFINED AND lastOnStatus <> _statusDualInput.STATUS_ERROR)) THEN
  			strKr.sdvig   := TRUE;
  		END_IF;
  	END_IF;
  END_IF;

  IF getSdvig THEN strKr.sdvig:= TRUE; END_IF;

  sdvigReset(IN:=strKr.sdvig, PT:=T#15S);

  IF sdvigReset.Q THEN strKr.sdvig:=FALSE; END_IF;

  lastOnStatus := strKr.onStatus;

  (* ---- Распаковка команды ---- *)
  _sunpackerCommand(command := strKr.inCommand);
  	cmd := _sunpackerCommand.cmd;
  	source := _sunpackerCommand.source;

  (* ---- Обработка команды ---- *)
  IF cmd <> 0 AND lastCmd <> cmd and (((NOT strKr.opcCommandsDisabled) AND source > 0) OR source = 0) then
  	CASE BYTE_TO_INT(cmd) OF
  	(*cmd_open*) 1 :
  			IF NOT BlockedOpenControl THEN
                                IF  strKr.ISVALIDREF_cmdOn THEN strKr.CmdOn := TRUE;
  				IF strKr.ISVALIDREF_cmdOff THEN strKr.CmdOff := FALSE; END_IF;
  			ELSIF  strKr.ISVALIDREF_cmdOff THEN strKr.CmdOff := FALSE;  END_IF;
  			errorCMDTimer(IN := false);

  			_commandErrorTimer := true;
  			strKr.lastCmdIsOn := true;
                                END_IF;
  	(*cmd_close*) 2 :
  			IF strKr.ISVALIDREF_cmdOff THEN strKr.CmdOff := TRUE;
  				IF strKr.ISVALIDREF_cmdOn THEN strKr.CmdOn := FALSE; END_IF;
  			ELSIF strKr.ISVALIDREF_cmdOn THEN strKr.CmdOn := FALSE; END_IF;
  			errorCMDTimer(IN := false);

  			_commandErrorTimer := true;
  			strKr.lastCmdIsOn := false;
  	(*cmd_reset*) 3 :   IF (strKr.ISVALIDREF_statOn) OR (strKr.ISVALIDREF_statOff) THEN
  			strKr.CmdOn := FALSE;
  			strKr.CmdOff := FALSE;
                                lastCmd := 0;
  			_commandErrorTimer := false;
  			strKr.lastCmdIsOn := false;
                                END_IF;

  	END_CASE;
  	source_for_Status := source;
  	cmd_for_Status := cmd;
  	command_error_for_Status := 0;
  END_IF;
  lastCmd := cmd;

  errorCMDTimer(In := _commandErrorTimer, PT :=T#90s);

  continueHoldCommandTimer(IN:=(strKr.onStatus = _statusDualInput.STATUS_ON) OR
  (strKr.onStatus = _statusDualInput.STATUS_OFF), PT:=strKr.continueHoldCommand);

  (* ---- алгоритм  для команды ВКЛючить ---- *)
  IF (strKr.onStatus = _statusDualInput.STATUS_ON) and strKr.lastCmdIsOn  then
  	IF strKr.ISVALIDREF_cmdOn AND strKr.ISVALIDREF_cmdOff then
            IF continueHoldCommandTimer.Q THEN
            strKr.cmdOn := false; END_IF;
            END_IF;
  	 errorCMDTimer(In := false);
  	 _commandErrorTimer := false;
  	 cmd_for_Status := 0;
  	 source_for_Status := 0;
  END_IF;

  (* ---- off ---- *)
  IF (strKr.onStatus = _statusDualInput.STATUS_OFF) and  (NOT strKr.lastCmdIsOn) then
  	IF strKr.ISVALIDREF_cmdOn AND strKr.ISVALIDREF_cmdOff then
            IF continueHoldCommandTimer.Q THEN
            strKr.cmdOff := false; END_IF;
            END_IF;
  	 errorCMDTimer(In := false);
  	 _commandErrorTimer := false;
  	 cmd_for_Status := 0;
  	 source_for_Status := 0;
  END_IF;

  (* ---- ошибка исполнения команды ---- *)
  if errorCMDTimer.Q and (cmd_for_Status <> 0) then
  	command_error_for_Status :=  cmd_for_Status;
  	_commandErrorTimer := false;
  	strKr.CmdOn := false;
  	strKr.CmdOff := false;
  	(*lastCmd := 0;*)
  END_IF;

  (* ---- сброс ошибки команды ---- *)
  strKr.CommandFault := command_error_for_Status <> 0;
  _errorReset(IN := command_error_for_Status <> 0, PT := T#5S);
  IF _errorReset.Q THEN
  	cmd_for_Status := 0;
  	source_for_Status := 0;
  	command_error_for_Status := 0;

  END_IF;

  outputsSets(in := (strKr.ISVALIDREF_cmdOn and strKr.cmdOn ) OR (strKr.ISVALIDREF_cmdOff and strKr.cmdOff), PT := T#2S);
  	IF NOT outputsSets.Q THEN
  		strKr.So := inSo._inversed AND inSo.reliability AND strKr.ISVALIDREF_inSo;
  		strKr.Sz := inSz._inversed AND inSz.reliability AND strKr.ISVALIDREF_inSz;
  	END_IF;

  cmdOn := strKr.cmdOn;
  cmdOff:= strKr.cmdOff;

  (* ---- формирование зашифрованного статуса для АРМа ---- *)
  strKr.status := shl(BYTE_TO_DWORD(source_for_Status), 29)
  		OR shl(BYTE_TO_DWORD(cmd_for_Status), 26)
  		OR shl(BYTE_TO_DWORD(command_error_for_Status), 23)
  		OR shl(bool_to_DWORD(strKr.sdvig), 22)
  		OR shl(bool_to_DWORD(strKr.OpcCommandsDisabled), 21)
                      OR shl(bool_to_DWORD(strKr.Dp), 14)
                      OR shl(BOOL_TO_DWORD(strKr.Sz), 13)
  		OR shl(BOOL_TO_DWORD(strKr.So), 12)
  		OR shl(BOOL_TO_DWORD(strKr.ErrorBlock), 11)
  		OR shl(BOOL_TO_DWORD(strKr.ErrorPowerOff), 10)
  		OR shl(BOOL_TO_DWORD(strKr.Manual), 8)
  		OR shl(BOOL_TO_DWORD(strKr.Auto), 7)
  		OR shl(BOOL_TO_DWORD(strKr.Distance), 6)
  		OR shl(BOOL_TO_DWORD(strKr.Local), 5)
  		OR shl(BOOL_TO_DWORD(strKr.Ns), 4)
                  	OR shl(BOOL_TO_DWORD(strKr.Accident ),3)
  		OR BYTE_TO_DWORD(strKr.onStatus);
END_FUNCTION_BLOCK

FUNCTION_BLOCK fb_DualStateIm
  VAR_INPUT
    statOn : BOOL;
    statOff : BOOL;
  END_VAR
  VAR_IN_OUT
    StrDs : struct_DualStateIm;
  END_VAR
  VAR_INPUT
    statOn_reliability : BOOL;
    statOff_reliability : BOOL;
    inNs : TYPE_ReliableBit;
    inAccident : TYPE_ReliableBit;
    inCommand : WORD;
  END_VAR
  VAR
    _statOn : BOOL;
    _statOff : BOOL;
    getSdvig : BOOL;
    lastOnStatus : BYTE;
    cmd : BYTE;
    source : BYTE;
    lastCmd : BYTE;
    source_for_Status : BYTE;
    cmd_for_Status : BYTE;
    command_error_for_Status : BYTE;
    _sunpackerCommand : fb_sunpackerCommand;
    _statusDualInput : TYPE_statusDualInput;
    _commandDualInput : TYPE_commandDualInput;
    _commandErrorTimer : BOOL;
    onInit : BOOL          := FALSE;
    resetErrorTimer : BOOL;
    _changWithoutCommand : BOOL;
    errorCMDTimer : TON;
    sdvigReset : TON;
    _errorReset : TON;
  END_VAR
  VAR_IN_OUT
    cmdOn : BOOL;
  END_VAR
  VAR_OUTPUT
    cmdOff : BOOL;
  END_VAR

  IF NOT onInit THEN
  IF StrDs.ISVALIDREF_cmdOn XOR StrDs.ISVALIDREF_cmdOff THEN
  	IF 	StrDs.ISVALIDREF_cmdOn THEN
  		lastCmd:= 2; (*baseCmdOff*)
  	ELSE
  		lastCmd:= 1; (*baseCmdOn*)
  	END_IF;
  END_IF;
  onInit:=TRUE;
  END_IF;

  (* ---- Если управление с ВУ заблокировано, то в ИМ передаем команду из алгоритма ---- *)
  IF StrDs.inOpcCommandsDisabled THEN
  	StrDs.inCommand := StrDs.inCommand_Alg;
  ELSE (* иначе передаем команду с АРМа*)
  	StrDs.inCommand := StrDs.inCommand_ARM;
  END_IF;

  (* ---- Формирование состояния механизма ---- *)

  IF (StrDs.ISVALIDREF_statOn) OR (StrDs.ISVALIDREF_statOff) THEN
  	IF (StrDs.ISVALIDREF_statOn) AND (StrDs.ISVALIDREF_statOff) THEN
  	StrDs.reliability:= statOn_reliability AND statOff_reliability;
  		_statOn  := statOn;
  		_statOff := statOff;
  	ELSIF (StrDs.ISVALIDREF_statOn) THEN
                       StrDs.reliability:= statOn_reliability;
  		_statOn  := statOn;
  		_statOff := NOT statOn;
  	ELSIF (StrDs.ISVALIDREF_statOff) THEN
  		 StrDs.reliability:= statOff_reliability;
  		_statOn  := NOT statOff;
  		_statOff :=statOff;
  	END_IF;

  	IF StrDs.reliability THEN
  		IF _statOn AND NOT _statOff 		THEN 	StrDs.onStatus := _statusDualInput.STATUS_ON;
  		ELSIF _statOff AND NOT _statOn 	THEN 	StrDs.onStatus := _statusDualInput.Status_OFF;
  		ELSIF NOT _statOn AND NOT _statOff 	THEN 	StrDs.onStatus := _statusDualInput.STATUS_TRANSITIONAL;
  		ELSE					StrDs.onStatus := _statusDualInput.STATUS_ERROR;
                      END_IF;

  	ELSE
  		StrDs.onStatus := _statusDualInput.STATUS_NOTDEFINED;

  	END_IF;
  ELSE
  	CASE BYTE_TO_INT(lastCmd) OF
  		(*baseCmdOn*) 1: StrDs.onStatus  := _statusDualInput.STATUS_ON;
  		(*baseCmdOff*) 2: StrDs.onStatus  := _statusDualInput.STATUS_OFF;

  	ELSE
  		 StrDs.onStatus := _statusDualInput.STATUS_NOTDEFINED;

  	END_CASE;
  END_IF;

  (* ---- Формирование признака сдвига ---- *)
  getSdvig := FALSE;
  IF (StrDs.ISVALIDREF_cmdOn OR StrDs.ISVALIDREF_cmdOff) THEN
  	IF NOT (StrDs.CmdOn OR StrDs.CmdOff) THEN
                       IF (lastOnStatus <> StrDs.onStatus AND
  		(StrDs.onStatus <> _statusDualInput.STATUS_NOTDEFINED AND
                       StrDs.onStatus <> _statusDualInput.STATUS_ERROR)     AND
  		(lastOnStatus <> _statusDualInput.STATUS_NOTDEFINED   AND
                       lastOnStatus <> _statusDualInput.STATUS_ERROR))
                      THEN
  			getSdvig   := TRUE;
  		END_IF;
  	END_IF;
  END_IF;

  IF getSdvig THEN StrDs.sdvig:= TRUE; END_IF;

  sdvigReset(IN:=StrDs.sdvig, PT:=T#15S);

  IF sdvigReset.Q THEN StrDs.sdvig:=FALSE; END_IF;

  lastOnStatus := StrDs.onStatus;

  StrDs.Accident := inAccident.value AND inAccident.reliability;
  StrDs.Ns := inNs.value AND inNs.reliability;
  StrDs.OpcCommandsDisabled := StrDs.inOpcCommandsDisabled;

  (* ---- Распаковка команды ---- *)
  _sunpackerCommand(command := StrDs.inCommand);
  	cmd := _sunpackerCommand.cmd;
  	source := _sunpackerCommand.source;

  (* ---- Обработка команды ---- *)
  IF cmd <> 0 AND lastCmd <> cmd and (((NOT StrDs.opcCommandsDisabled) AND source > 0) OR source = 0) then
  	CASE BYTE_TO_INT(cmd) OF
  	(*cmd_open*) 1 :
  			IF  StrDs.ISVALIDREF_cmdOn THEN StrDs.CmdOn := TRUE;
  				IF StrDs.ISVALIDREF_cmdOff THEN StrDs.CmdOff := FALSE; END_IF;
  			ELSIF  StrDs.ISVALIDREF_cmdOff THEN StrDs.CmdOff := FALSE;  END_IF;
  			errorCMDTimer(IN := false);
  			_commandErrorTimer := true;
  			StrDs.lastCmdIsOn := true;
  	(*cmd_close*) 2 :
  			IF StrDs.ISVALIDREF_cmdOff THEN StrDs.CmdOff := TRUE;
  				IF StrDs.ISVALIDREF_cmdOn THEN StrDs.CmdOn := FALSE; END_IF;
  			ELSIF StrDs.ISVALIDREF_cmdOn THEN StrDs.CmdOn := FALSE; END_IF;
  			errorCMDTimer(IN := false);
  			_commandErrorTimer := true;
  			StrDs.lastCmdIsOn := false;
  	(*cmd_reset*) 3 :    IF StrDs.ISVALIDREF_statOn OR StrDs.ISVALIDREF_statOff THEN
  			StrDs.CmdOn := FALSE;
  			StrDs.CmdOff := FALSE;
                                lastCmd :=0;
  			_commandErrorTimer := false;
  			StrDs.lastCmdIsOn := false;
                                END_IF;
  	END_CASE;
  	source_for_Status := source;
  	cmd_for_Status := cmd;
  	command_error_for_Status := 0;
  END_IF;

  lastCmd := cmd;
  errorCMDTimer(In := _commandErrorTimer, PT :=T#10s);

  (* ---- алгоритм  для команды ВКЛючить ---- *)
  IF (StrDs.onStatus = _statusDualInput.STATUS_ON) and (lastCmd = _commandDualInput.CMD_ON) then
  	IF StrDs.ISVALIDREF_cmdOn AND StrDs.ISVALIDREF_cmdOff then  StrDs.cmdOn := false; END_IF;

  	 errorCMDTimer(In := false);
  	 _commandErrorTimer := false;
  	 cmd_for_Status := 0;
  	 source_for_Status := 0;
  END_IF;

  (* ---- off ---- *)
  IF (StrDs.onStatus = _statusDualInput.STATUS_OFF) and (lastCmd = _commandDualInput.CMD_OFF) then
  	IF StrDs.ISVALIDREF_cmdOn AND StrDs.ISVALIDREF_cmdOff then  StrDs.cmdOff := false; END_IF;

  	 errorCMDTimer(In := false);
  	 _commandErrorTimer := false;
  	 cmd_for_Status := 0;
  	 source_for_Status := 0;
  END_IF;

  (* ---- ошибка исполнения команды ---- *)
  if errorCMDTimer.Q and (cmd_for_Status <> 0) then
  	command_error_for_Status :=  cmd_for_Status;
  	_commandErrorTimer := false;
  	StrDs.CmdOn := false;
  	StrDs.CmdOff := false;
  	lastCmd := 0;
  end_if;

  (* ---- сброс ошибки команды ---- *)
  StrDs.CommandFault := command_error_for_Status <> 0;
  _errorReset(IN := command_error_for_Status <> 0, PT := T#15S);
  IF _errorReset.Q THEN
  	cmd_for_Status := 0;
  	source_for_Status := 0;
  	command_error_for_Status := 0;
  END_IF;

  cmdOn := StrDs.cmdOn;
  cmdOff:= StrDs.cmdOff;

  (* ---- формирование зашифрованного статуса для АРМа ---- *)
  StrDs.status := shl(BYTE_TO_DWORD(source_for_Status), 29)
  		OR shl(BYTE_TO_DWORD(cmd_for_Status), 26)
  		OR shl(BYTE_TO_DWORD(command_error_for_Status), 23)
  		OR shl(bool_to_DWORD(StrDs.sdvig), 22)
  		OR shl(bool_to_DWORD(StrDs.OpcCommandsDisabled), 21)
  		OR shl(BOOL_TO_DWORD(StrDs.Ns), 4)
                  	OR shl(BOOL_TO_DWORD(StrDs.Accident ),3)
  		OR BYTE_TO_DWORD(StrDs.onStatus);
END_FUNCTION_BLOCK

FUNCTION_BLOCK fb_AO_Init
  VAR_INPUT
    data_Ini : BOOL;
    outLL : LREAL          := 4000.0;
    outHL : LREAL          := 20000.0;
    newLL : LREAL;
    newHL : LREAL;
    newLL_ISVALIDREF : BOOL;
    newHL_ISVALIDREF : BOOL;
  END_VAR
  VAR_IN_OUT
    strAO : struct_AO;
  END_VAR
  VAR_OUTPUT
    Init : BOOL          := FALSE;
  END_VAR

  (*****            Функциональный блок переинициализации структуры-дескриптора канала аналогового ввода.            *****)

   Init := FALSE;

      IF data_Ini THEN                            (* Параметрам требуется переинициализация. *)
          strAO.outLL                := outLL;
          strAO.outHL                := outHL;
          strAO.newLL                := newLL;
          strAO.newHL                := newHL;
          strAO.newLL_ISVALIDREF     := newLL_ISVALIDREF;
          strAO.newHL_ISVALIDREF     := newHL_ISVALIDREF;
          data_Ini:=FALSE;
          Init := TRUE;
      END_IF;
   IF Init THEN
         (* outLL:=0.0;*)
         (* outHL:=0.0;*)
          newLL:=0.0;
          newHL:=0.0;
          newLL_ISVALIDREF:= FALSE;
          newHL_ISVALIDREF:= FALSE;
   END_IF;
END_FUNCTION_BLOCK

FUNCTION_BLOCK fb_DiProtection
  VAR_INPUT
    di : struct_singleSignal;
  END_VAR
  VAR_IN_OUT
    StrDIp : struct_DiProtection;
  END_VAR
  VAR
    _sunpackerCommand : fb_sunpackerCommand;
    _ProtectionTags : TYPE_ProtectionTags;
    _signalingTp : TOF;
    timer : TON;
    SignalingTrig : R_TRIG;
    SignalingFTrig : F_TRIG;
    SignalingDi : BOOL;
    source : BYTE;
    cmd : BYTE;
    lastCmd : BYTE;
    source_for_Status : BYTE;
    cmd_for_Status : BYTE;
    command_error_for_Status : BYTE;
    resetCmdTimer : TON;
    resetCmdTimerPriznak : BOOL;
    signalinTimer : TON;
    runOnStart_Trig : R_TRIG;
  END_VAR

  timer(IN := di.Q AND StrDIp.isRunning  , PT := StrDIp.delay);
  SignalingTrig(CLK := timer.Q);
  IF SignalingTrig.Q THEN
  	SignalingDi := TRUE;
  END_IF;
  SignalingFTrig(CLK := timer.Q);
  IF SignalingFTrig.Q THEN
  	SignalingDi := FALSE;
  END_IF;

  StrDIp.Tag := StrDIp.inTag;
  StrDIp.RunOnStart := StrDIp.inRunOnStart;

  StrDIp.CanRun := StrDIp.inCanRun;

  StrDIp.OpcCommandsDisabled := StrDIp.inOpcCommandsDisabled;

  (* ---- Если управление с ВУ заблокировано, то передаем команду из алгоритма ---- *)
  IF StrDIp.inOpcCommandsDisabled THEN
  	StrDIp.inCommand := StrDIp.inCommand_Alg;
  ELSE (* иначе передаем команду с АРМа*)
  	StrDIp.inCommand := StrDIp.inCommand_ARM;
  END_IF;

  _sunpackerCommand(command := StrDIp.inCommand);
  	source := _sunpackerCommand.source;
  	cmd := _sunpackerCommand.cmd;

  IF cmd <> 0 AND lastCmd <> cmd AND (((NOT StrDIp.opcCommandsDisabled) AND source > 0) OR source = 0) then

  	CASE BYTE_TO_INT(cmd) OF
  	        (*cmdRun*) 1: 	IF        NOT StrDIp.Remont THEN
  					StrDIp.isEnded := FALSE;
  					StrDIp.hasError 	:= FALSE;
  					StrDIp.isRunning := TRUE;
  					cmd_for_Status := cmd;
  					source_for_Status := source;
  					command_error_for_Status := 0;
  				ELSE
  					StrDIp.isRunning := FALSE;
  					StrDIp.isEnded := FALSE;
  					StrDIp.hasError 	:= FALSE;

  					cmd_for_Status := 0;
  					source_for_Status := source;
  					command_error_for_Status := cmd;
  				END_IF;
                                          StrDIp.inOpcCommandsDisabled:=FALSE;

                  (*cmdReset*) 2: 	StrDIp.isRunning := FALSE;
  				StrDIp.isEnded := FALSE;
  				StrDIp.hasError 	:= FALSE;
  				SignalingDi:= FALSE;
  				StrDIp.Check := FALSE;
  				cmd_for_Status := cmd;
  				source_for_Status := source;
  				command_error_for_Status := 0;
                                         StrDIp.inOpcCommandsDisabled:=FALSE;

  	(*cmd_setRemont*) 4 :	StrDIp.Remont := TRUE;
  				(*StrDIp.isRunning := FALSE;*)

  				cmd_for_Status := cmd;
  				source_for_Status := source;
  				command_error_for_Status := 0;
          (*cmd_resetRemont*) 5 : 	(*IF di.Q THEN
  					cmd_for_Status := 0;
  					source_for_Status := 0;
  					command_error_for_Status := cmd;
  				ELSE*)
  					StrDIp.Remont := FALSE;
  					(*StrDIp.isRunning := TRUE;*)

  					cmd_for_Status := cmd;
  					source_for_Status := source;
  					command_error_for_Status := 0;
  				(*END_IF;*)
  	(*cmd_setCheck*) 6 : 	StrDIp.Check := TRUE;

  				cmd_for_Status := cmd;
  				source_for_Status := source;
  				command_error_for_Status := 0;
  	END_CASE;
  	resetCmdTimer(IN := false);
  	resetCmdTimerPriznak := TRUE;
  END_IF;
  lastCmd := cmd;

  resetCmdTimer(IN := resetCmdTimerPriznak);
  IF resetCmdTimer.Q THEN
  	resetCmdTimerPriznak := FALSE;
  	source_for_Status := 0;
  	cmd_for_Status := 0;
  	command_error_for_Status := 0;
  END_IF;

  IF StrDIp.isRunning AND NOT StrDIp.Remont AND NOT StrDIp.Check THEN
  	StrDIp.Signaling := SignalingDi;
  	StrDIp.SignalingTP := _signalingTp.Q;
  ELSE
  	StrDIp.Signaling := 0;
  	StrDIp.SignalingTP := 0;
  END_IF;

  _signalingTp(in := StrDIp.Signaling, PT := T#1s);

  StrDIp.status :=  SHL(BYTE_TO_DWORD(source_for_Status), 29)
  			OR SHL(BYTE_TO_DWORD(cmd_for_Status), 26)
  			OR SHL(BYTE_TO_DWORD(command_error_for_Status), 23)
  			OR SHL(BOOL_TO_DWORD(StrDIp.OpcCommandsDisabled ), 21)
  			OR SHL(BOOL_TO_DWORD(StrDIp.Signaling), 16)
  			OR SHL(BOOL_TO_DWORD(StrDIp.RunOnStart ), 15)
  			OR SHL(BOOL_TO_DWORD(StrDIp.remont), 6)
  			OR SHL(BOOL_TO_DWORD(StrDIp.Check), 5)
  			OR SHL(BOOL_TO_DWORD(StrDIp.hasError), 4)
  			OR SHL(BOOL_TO_DWORD(StrDIp.SignalingTP), 3)
  			OR SHL(BOOL_TO_DWORD(StrDIp.CanRun), 2)
  			OR SHL(BOOL_TO_DWORD(StrDIp.isEnded), 1)
  			OR BOOL_TO_DWORD(StrDIp.isRunning);
END_FUNCTION_BLOCK

FUNCTION_BLOCK fb_KranOpenProtection
  VAR_INPUT
    im : struct_Kran;
  END_VAR
  VAR_IN_OUT
    StrDIp : struct_DiProtection;
  END_VAR
  VAR
    _sunpackerCommand : fb_sunpackerCommand;
    statusDualInput : TYPE_statusDualInput;
    _ProtectionTags : TYPE_ProtectionTags;
    _signalingTp : TOF;
    timer : TON;
    SignalingTrig : R_TRIG;
    SignalingFTrig : F_TRIG;
    SignalingDi : BOOL;
    source : BYTE;
    cmd : BYTE;
    lastCmd : BYTE;
    source_for_Status : BYTE;
    cmd_for_Status : BYTE;
    command_error_for_Status : BYTE;
    resetCmdTimer : TON;
    resetCmdTimerPriznak : BOOL;
    signalinTimer : TON;
    runOnStart_Trig : R_TRIG;
  END_VAR

  timer(IN := (im.onStatus<>statusDualInput.STATUS_ON) AND StrDIp.isRunning  , PT := StrDIp.delay);
  SignalingTrig(CLK := timer.Q);
  IF SignalingTrig.Q THEN
  	SignalingDi := TRUE;
  END_IF;
  SignalingFTrig(CLK := timer.Q);
  IF SignalingFTrig.Q THEN
  	SignalingDi := FALSE;
  END_IF;

  StrDIp.Tag := StrDIp.inTag;
  StrDIp.RunOnStart := StrDIp.inRunOnStart;

  StrDIp.CanRun := StrDIp.inCanRun;

  StrDIp.OpcCommandsDisabled := StrDIp.inOpcCommandsDisabled;

  (* ---- Если управление с ВУ заблокировано, то передаем команду из алгоритма ---- *)
  IF StrDIp.inOpcCommandsDisabled THEN
  	StrDIp.inCommand := StrDIp.inCommand_Alg;
  ELSE (* иначе передаем команду с АРМа*)
  	StrDIp.inCommand := StrDIp.inCommand_ARM;
  END_IF;

  _sunpackerCommand(command := StrDIp.inCommand);
  	source := _sunpackerCommand.source;
  	cmd := _sunpackerCommand.cmd;

  IF cmd <> 0 AND lastCmd <> cmd AND (((NOT StrDIp.opcCommandsDisabled) AND source > 0) OR source = 0) then
  	CASE BYTE_TO_INT(cmd) OF
  	        (*cmdRun*) 1: 	IF        NOT StrDIp.Remont THEN
  					StrDIp.isEnded := FALSE;
  					StrDIp.hasError 	:= FALSE;
  					StrDIp.isRunning := TRUE;
  					cmd_for_Status := cmd;
  					source_for_Status := source;
  					command_error_for_Status := 0;
  				ELSE
  					StrDIp.isRunning := FALSE;
  					StrDIp.isEnded := FALSE;
  					StrDIp.hasError 	:= FALSE;

  					cmd_for_Status := 0;
  					source_for_Status := source;
  					command_error_for_Status := cmd;
  				END_IF;
                                          StrDIp.inOpcCommandsDisabled:=FALSE;

                  (*cmdReset*) 2: 	StrDIp.isRunning := FALSE;
  				StrDIp.isEnded := FALSE;
  				StrDIp.hasError 	:= FALSE;
  				SignalingDi:= FALSE;
  				StrDIp.Check := FALSE;
  				cmd_for_Status := cmd;
  				source_for_Status := source;
  				command_error_for_Status := 0;
                                          StrDIp.inOpcCommandsDisabled:=FALSE;

  	(*cmd_setRemont*) 4 :	StrDIp.Remont := TRUE;
  				(*StrDIp.isRunning := FALSE;*)

  				cmd_for_Status := cmd;
  				source_for_Status := source;
  				command_error_for_Status := 0;

          (*cmd_resetRemont*) 5 : 	(*IF (im.onStatus<>statusDualInput.STATUS_ON) THEN
  					cmd_for_Status := 0;
  					source_for_Status := 0;
  					command_error_for_Status := cmd;
  				ELSE*)
  					StrDIp.Remont := FALSE;
  					(*StrDIp.isRunning := TRUE;*)

  					cmd_for_Status := cmd;
  					source_for_Status := source;
  					command_error_for_Status := 0;
  				(*END_IF;*)

  	(*cmd_setCheck*) 6 : 	StrDIp.Check := TRUE;

  				cmd_for_Status := cmd;
  				source_for_Status := source;
  				command_error_for_Status := 0;
  	END_CASE;
  	resetCmdTimer(IN := false);
  	resetCmdTimerPriznak := TRUE;
  END_IF;
  lastCmd := cmd;

  resetCmdTimer(IN := resetCmdTimerPriznak);
  IF resetCmdTimer.Q THEN
  	resetCmdTimerPriznak := FALSE;
  	source_for_Status := 0;
  	cmd_for_Status := 0;
  	command_error_for_Status := 0;
  END_IF;

  IF StrDIp.isRunning AND  NOT StrDIp.Remont AND NOT StrDIp.Check THEN
  	StrDIp.Signaling := SignalingDi;
  	StrDIp.SignalingTP := _signalingTp.Q;
  ELSE
  	StrDIp.Signaling := 0;
  	StrDIp.SignalingTP := 0;
  END_IF;

  _signalingTp(in := StrDIp.Signaling, PT := T#1s);

  StrDIp.status :=  SHL(BYTE_TO_DWORD(source_for_Status), 29)
  			OR SHL(BYTE_TO_DWORD(cmd_for_Status), 26)
  			OR SHL(BYTE_TO_DWORD(command_error_for_Status), 23)
  			OR SHL(BOOL_TO_DWORD(StrDIp.OpcCommandsDisabled ), 21)
  			OR SHL(BOOL_TO_DWORD(StrDIp.Signaling), 16)
  			OR SHL(BOOL_TO_DWORD(StrDIp.RunOnStart ), 15)
  			OR SHL(BOOL_TO_DWORD(StrDIp.remont), 6)
  			OR SHL(BOOL_TO_DWORD(StrDIp.Check), 5)
  			OR SHL(BOOL_TO_DWORD(StrDIp.hasError), 4)
  			OR SHL(BOOL_TO_DWORD(StrDIp.SignalingTP), 3)
  			OR SHL(BOOL_TO_DWORD(StrDIp.CanRun), 2)
  			OR SHL(BOOL_TO_DWORD(StrDIp.isEnded), 1)
  			OR BOOL_TO_DWORD(StrDIp.isRunning);
END_FUNCTION_BLOCK

FUNCTION_BLOCK fb_AiProtection
  VAR_INPUT
    ai : struct_AI;
  END_VAR
  VAR_IN_OUT
    StrAIp : struct_AiProtection;
  END_VAR
  VAR
    _sunpackerCommand : fb_sunpackerCommand;
    _signalingTp : TOF;
    _statusAi : TYPE_StatusAi;
    source : BYTE;
    cmd : BYTE;
    lastCmd : BYTE;
    source_for_Status : BYTE;
    cmd_for_Status : BYTE;
    command_error_for_Status : BYTE;
    resetCmdTimer : TON;
    resetCmdTimerPriznak : BOOL;
    signalinTimer : TON;
    timer : TON;
    SignalingTrig : R_TRIG;
    SignalingFTrig : F_TRIG;
    SignalingAi : BOOL;
  END_VAR

  timer(IN :=(ai.interval=StrAIp.controlLimit) AND (ai.interval >= _statusAi.normal) AND StrAIp.isRunning, PT :=StrAIp.delay);
  SignalingTrig(CLK := timer.Q);
  IF SignalingTrig.Q THEN
  	SignalingAi := TRUE;
  END_IF;
  SignalingFTrig(CLK := timer.Q);
  IF SignalingFTrig.Q THEN
  	SignalingAi := FALSE;
  END_IF;

  StrAIp.Tag := StrAIp.inTag;
  StrAIp.RunOnStart := StrAIp.inRunOnStart;

  StrAIp.CanRun := StrAIp.inCanRun;

  StrAIp.OpcCommandsDisabled := StrAIp.inOpcCommandsDisabled;

  (* ---- Если управление с ВУ заблокировано, то передаем команду из алгоритма ---- *)
  IF StrAIp.inOpcCommandsDisabled THEN
  	StrAIp.inCommand := StrAIp.inCommand_Alg;
  ELSE (* иначе передаем команду с АРМа*)
  	StrAIp.inCommand := StrAIp.inCommand_ARM;
  END_IF;

  _sunpackerCommand(command := StrAIp.inCommand);
  	source := _sunpackerCommand.source;
  	cmd := _sunpackerCommand.cmd;

  IF cmd <> 0 AND lastCmd <> cmd AND (((NOT StrAIp.opcCommandsDisabled) AND source > 0) OR source = 0) then

  	CASE BYTE_TO_INT(cmd) OF
  		(*cmdRun*) 1: 	IF        NOT StrAIp.Remont THEN
  					StrAIp.isEnded := FALSE;
  					StrAIp.hasError 	:= FALSE;
  					StrAIp.isRunning := TRUE;

  					cmd_for_Status := cmd;
  					source_for_Status := source;
  					command_error_for_Status := 0;
  				ELSE
  					StrAIp.isRunning := FALSE;
  					StrAIp.isEnded := FALSE;
  					StrAIp.hasError 	:= FALSE;

  					cmd_for_Status := 0;
  					source_for_Status := source;
  					command_error_for_Status := cmd;
  				END_IF;
                                          StrAIp.inopcCommandsDisabled:=FALSE;

  		(*cmdReset*) 2: 	StrAIp.isRunning := FALSE;
  				StrAIp.isEnded := FALSE;
  				StrAIp.hasError 	:= FALSE;
  				SignalingAi := FALSE;
  				StrAIp.Check := FALSE;
                                          (*StrAIp.Remont := FALSE;*)
  				cmd_for_Status := cmd;
  				source_for_Status := source;
  				command_error_for_Status := 0;
                                          StrAIp.inopcCommandsDisabled:=FALSE;

  	(*cmd_setRemont*) 4 :	StrAIp.Remont := TRUE;
  				(*StrAIp.isRunning := FALSE;*)

  				cmd_for_Status := cmd;
  				source_for_Status := source;
  				command_error_for_Status := 0;
  	(*cmd_resetRemont*) 5 : 	(*IF (ai.interval=StrAIp.controlLimit) THEN
  					cmd_for_Status := 0;
  					source_for_Status := 0;
  					command_error_for_Status := cmd;
  				ELSE*)
  					StrAIp.Remont := FALSE;
  					(*StrAIp.isRunning := TRUE;*)

  					cmd_for_Status := cmd;
  					source_for_Status := source;
  					command_error_for_Status := 0;
  				(*END_IF;*)
  	(*cmd_setCheck*) 6 : 	StrAIp.Check := TRUE;

  				cmd_for_Status := cmd;
  				source_for_Status := source;
  				command_error_for_Status := 0;
  	END_CASE;
  	resetCmdTimer(IN := false);
  	resetCmdTimerPriznak := TRUE;
  END_IF;
  lastCmd := cmd;

  resetCmdTimer(IN := resetCmdTimerPriznak);
  IF resetCmdTimer.Q THEN
  	resetCmdTimerPriznak := FALSE;
  	source_for_Status := 0;
  	cmd_for_Status := 0;
  	command_error_for_Status := 0;
  END_IF;

  IF StrAIp.isRunning AND NOT StrAIp.Remont AND NOT StrAIp.Check THEN
  	StrAIp.Signaling := SignalingAi;
  	StrAIp.SignalingTP := _signalingTp.Q;
  ELSE
  	StrAIp.Signaling := 0;
  	StrAIp.SignalingTP := 0;
  END_IF;

  _signalingTp(in := StrAIp.Signaling, PT := T#1s);

  StrAIp.status :=  SHL(BYTE_TO_DWORD(source_for_Status), 29)
  			OR SHL(BYTE_TO_DWORD(cmd_for_Status), 26)
  			OR SHL(BYTE_TO_DWORD(command_error_for_Status), 23)
  			OR SHL(BOOL_TO_DWORD(StrAIp.OpcCommandsDisabled ), 21)
  			OR SHL(BOOL_TO_DWORD(StrAIp.Signaling), 16)
  			OR SHL(BOOL_TO_DWORD(StrAIp.RunOnStart ), 15)
  			OR SHL(BOOL_TO_DWORD(StrAIp.remont), 6)
  			OR SHL(BOOL_TO_DWORD(StrAIp.Check), 5)
  			OR SHL(BOOL_TO_DWORD(StrAIp.hasError), 4)
  			OR SHL(BOOL_TO_DWORD(StrAIp.SignalingTP), 3)
  			OR SHL(BOOL_TO_DWORD(StrAIp.CanRun), 2)
  			OR SHL(BOOL_TO_DWORD(StrAIp.isEnded), 1)
  			OR BOOL_TO_DWORD(StrAIp.isRunning);
END_FUNCTION_BLOCK

FUNCTION_BLOCK proc_Protection
  VAR
    fb_mvOff : fb_MvProtection;
    fb_dPmaslo_gaz_Less100 : fb_DiProtection;
    fb_Reg_vozb_off : fb_DiProtection;
    fb_Fail_chastotnii_pusk : fb_DiProtection;
    fb_Off_avar_vikluchatel : fb_DiProtection;
    fb_AOKC_SHKC : fb_DiProtection;
    fb_AO_PRU : fb_DiProtection;
    fb_AO_ot_SHU : fb_DiProtection;
    fb_Kran1_sdvig : fb_KranOpenProtection;
    fb_Kran2_sdvig : fb_KranOpenProtection;
    fb_Toporno_podshipnika_EDT_1 : fb_AiProtection;
    fb_Toy_podshipnika_EDT_2 : fb_AiProtection;
    fb_Toy_podshipnika_kol_EDT_3 : fb_AiProtection;
    fb_Toy_podshipnika_kol_EDT_4 : fb_AiProtection;
    fb_Toy_podshipnika_shest_red_EDT_5 : fb_AiProtection;
    fb_Ty_podshipnika_red_EDT_6 : fb_AiProtection;
    fb_Ty_podshipnika_nagnet_EDT_7_1 : fb_AiProtection;
    fb_Ty_podshipnika_nagnet_EDT_7_2 : fb_AiProtection;
    fb_Toy_podshipnika_svobod_konca_EDT_8_1 : fb_AiProtection;
    fb_Toy_podshipnika_svobod_konca_EDT_8_2 : fb_AiProtection;
    fb_Toy_podshipnika_rab_kol_EDT_9_1 : fb_AiProtection;
    fb_Toy_podshipnika_rab_kol_EDT_9_2 : fb_AiProtection;
    fb_Toy_podshipnika_nerab_kol_EDT_10_1 : fb_AiProtection;
    fb_Toy_podshipnika_nerab_kol_EDT_10_2 : fb_AiProtection;
    fb_Tgaza_na_vhode_H : fb_AiProtection;
    fb_Tgaza_na_vyhode_H : fb_AiProtection;
    fb_Tmasla_v_mb : fb_AiProtection;
    fb_Tmasla_v_mb_nad_ten : fb_AiProtection;
    fb_Tgorjachego_vozduha_ED_kanal_1 : fb_AiProtection;
    fb_Tgorjachego_vozduha_ED_kanal_2 : fb_AiProtection;
    fb_Tmasla_do_AVOM : fb_AiProtection;
    fb_Tmasla_posle_AVOM : fb_AiProtection;
    fb_Tmedi_statora_kanal_1 : fb_AiProtection;
    fb_Tmedi_statora_kanal_2 : fb_AiProtection;
    fb_Tmedi_statora_kanal_3 : fb_AiProtection;
    fb_Tstali_statora_kanal_1 : fb_AiProtection;
    fb_Tstali_statora_kanal_2 : fb_AiProtection;
    fb_Tstali_statora_kanal_3 : fb_AiProtection;
    fb_Tholodnogo_vozduha_ED_kanal_1 : fb_AiProtection;
    fb_Tholodnogo_vozduha_ED_kanal_2 : fb_AiProtection;
    fb_Pmaslo_sm_nizkoe : fb_AiProtection;
    fb_Pmaslo_sm_vysokoe : fb_AiProtection;
    fb_Pgaza_na_vhode_nagnetatelia : fb_AiProtection;
    fb_Pgaza_na_vyhode_nagnetatelia : fb_AiProtection;
    fb_Pmasla_posle_NU : fb_AiProtection;
    fb_Pmasla_smazki_posle_gns : fb_AiProtection;
    fb_Pimpuls_gaz : fb_AiProtection;
    fb_dPmaslo_gaz : fb_AiProtection;
    fb_dP_maslo_na_filtre : fb_AiProtection;
    fb_Os_sdvig_nagnetatelja_plus : fb_AiProtection;
    fb_Os_sdvig_nagnetatelja_minus : fb_AiProtection;
    fb_Vibro_skorost_OPED_T1 : fb_AiProtection;
    fb_Vibro_skorost_OPED_T2 : fb_AiProtection;
    fb_Vibro_skorost_OYP_kolesa_ED_T3 : fb_AiProtection;
    fb_Vibro_skorost_OP_kolesa_RH_T4 : fb_AiProtection;
    fb_Vibro_skorost_OP_shesterni_RED_T5 : fb_AiProtection;
    fb_Vibro_skorost_OP_shesterni_RED_T6 : fb_AiProtection;
    fb_Vibroperemesh_vala_N_T7 : fb_AiProtection;
    fb_Vibroperemesh_vala_N_T8 : fb_AiProtection;
    fb_Uroven_masla_v_mb : fb_AiProtection;
    fb_Tok_statora : fb_AiProtection;
    fb_Kontrol_per_220V_less187 : fb_AiProtection;
    fb_Kontrol_per_220V_high242 : fb_AiProtection;
    fb_Kontrol_post_220V_less187 : fb_AiProtection;
    fb_Kontrol_post_220V_high242 : fb_AiProtection;
  END_VAR
  VAR_EXTERNAL
    protections : ProtectionsConfig;
    ai : AiConfig;
    IM : ImConfig;
  END_VAR

  (************************************************************* DiProtection ************************************************************)
  (* МВ отключен
  fb_mvOff(sw:=IM.mv, StrDIp := protections.Pgaza_na_vyhode_nagnetatelia_GPA_STOP);*)

  (* Неисправность возбудительного устройства *)
  fb_dPmaslo_gaz_Less100(di := IM.SingleSignals.dP_maslo_gaz_Less100, StrDIp := protections.dPmaslo_gaz_less100);

  (* Сдвиг крана №2 *)
  fb_Reg_vozb_off(di:=IM.SingleSignals.Vozbud_neispravnost, StrDIp := protections.Reg_vozb_off);

  (* Сдвиг крана №2 *)
  fb_Fail_chastotnii_pusk(di:=IM.SingleSignals.Neuspesh_chastotny_pusk, StrDIp := protections.Fail_chastotnii_pusk);

  (* Сдвиг крана №2 *)
  fb_Off_avar_vikluchatel(di:=IM.SingleSignals.Avariinoe_otkluch_vikluchatelya, StrDIp := protections.Off_avar_vikluchatel);

  (* Сдвиг крана №2 *)
  fb_AOKC_SHKC(di:=IM.SingleSignals.AO_KC_ot_SHKS, StrDIp := protections.AOKC_SHKC);

  (* Сдвиг крана №2 *)
  fb_AO_PRU(di:=IM.SingleSignals.AO_GPA_ot_PRU, StrDIp := protections.AO_PRU);

  (* Сдвиг крана №2 *)
  fb_AO_ot_SHU(di:=IM.SingleSignals.AO_GPA_ot_SHU, StrDIp := protections.AO_ot_SHU);

  (* Сдвиг крана №2 *)
  fb_Kran1_sdvig(im:=IM.Kran1, StrDIp := protections.Kran1_sdvig);

  (* Сдвиг крана №2 *)
  fb_Kran2_sdvig(im:=IM.Kran2, StrDIp := protections.Kran2_sdvig);

  (************************************************************* AiProtection ************************************************************)

  (* Температура переднего опорного подшипника двигателя, т.1 *)
  fb_Toporno_podshipnika_EDT_1(ai := ai.Toporno_podshipnika_EDT_1, StrAIp := protections.Topornogo_podshipnika_EDT_1);

  (* Температура заднего опорного подшипника двигателя, т.2 *)
  fb_Toy_podshipnika_EDT_2(ai := ai.Toy_podshipnika_EDT_2, StrAIp := protections.Toy_podshipnika_EDT_2);

  (* Температура подшипника редуктора, т1 *)
  fb_Toy_podshipnika_kol_EDT_3(ai := ai.Toy_podshipnika_kol_EDT_3, StrAIp := protections.Toy_podshipnika_kol_EDT_3);

  (* Температура подшипника редуктора, т2 *)
  fb_Toy_podshipnika_kol_EDT_4(ai := ai.Toy_podshipnika_kol_EDT_4, StrAIp := protections.Toy_podshipnika_kol_EDT_4);

  (* Температура подшипника редуктора, т3 *)
  fb_Toy_podshipnika_shest_red_EDT_5(ai := ai.Toy_podshipnika_shest_red_EDT_5, StrAIp := protections.To_podshipnika_shest_red_EDT_5);

  (* Температура подшипника редуктора, т4 *)
  fb_Ty_podshipnika_red_EDT_6(ai := ai.Ty_podshipnika_red_EDT_6, StrAIp := protections.To_podshipnika_shest_red_EDT_6);

  (* Температура опорного подшипника нагнетателя, т1 *)
  fb_Ty_podshipnika_nagnet_EDT_7_1(ai := ai.Ty_podshipnika_nagnet_EDT_7_1, StrAIp := protections.To_podshipnika_N_EDT_7);

  (* Температура опорного подшипника нагнетателя, т1 *)
  fb_Ty_podshipnika_nagnet_EDT_7_2(ai := ai.Ty_podshipnika_nagnet_EDT_7_2, StrAIp := protections.To_podshipnika_N_EDT_7);

  (* Температура опорного подшипника нагнетателя, т2 *)
  fb_Toy_podshipnika_svobod_konca_EDT_8_1(ai := ai.Toy_podshipnika_svobod_konca_EDT_8_1, StrAIp := protections.To_podshipnika_svob_konca_EDT_8);

  (* Температура опорного подшипника нагнетателя, т2 *)
  fb_Toy_podshipnika_svobod_konca_EDT_8_2(ai := ai.Toy_podshipnika_svobod_konca_EDT_8_2, StrAIp := protections.To_podshipnika_svob_konca_EDT_8);

  (* Температура опорного подшипника нагнетателя, т3 *)
  fb_Toy_podshipnika_rab_kol_EDT_9_1(ai := ai.Toy_podshipnika_rab_kol_EDT_9_1, StrAIp := protections.Ty_podshipnika_rab_kol_EDT_9);

  (* Температура опорного подшипника нагнетателя, т3 *)
  fb_Toy_podshipnika_rab_kol_EDT_9_2(ai := ai.Toy_podshipnika_rab_kol_EDT_9_2, StrAIp := protections.Ty_podshipnika_rab_kol_EDT_9);

  (* Температура упорно опорного подшипника нагнетателя, т4 *)
  fb_Toy_podshipnika_nerab_kol_EDT_10_1(ai := ai.Toy_podshipnika_nerab_kol_EDT_10_1, StrAIp := protections.Typornogo_podshipnika_nerab_kolodok_HT_10);

  (* Температура упорно опорного подшипника нагнетателя, т4 *)
  fb_Toy_podshipnika_nerab_kol_EDT_10_2(ai := ai.Toy_podshipnika_nerab_kol_EDT_10_2, StrAIp := protections.Typornogo_podshipnika_nerab_kolodok_HT_10);

  (* Температура газа на выходе нагнетателя *)
  fb_Tgaza_na_vyhode_H(ai := ai.Tgaza_na_vhode_H, StrAIp := protections.Tgaza_na_vyhode_H);

  (* Температура газа на выходе нагнетателя *)
  fb_Os_sdvig_nagnetatelja_plus(ai := ai.Os_sdvig_nagnetatelja_plus, StrAIp := protections.Os_sdvig_nagnetatelja_plus);

  (* Температура газа на выходе нагнетателя *)
  fb_Os_sdvig_nagnetatelja_minus(ai := ai.Os_sdvig_nagnetatelja_minus, StrAIp := protections.Os_sdvig_nagnetatelja_minus);

  (* Температура газа на выходе нагнетателя *)
  fb_Pgaza_na_vyhode_nagnetatelia(ai := ai.Pgaza_na_vyhode_nagnetatelia, StrAIp := protections.Pgaza_na_vyhode_nagnetatelia);

  (* Температура газа на выходе нагнетателя *)
  fb_dPmaslo_gaz(ai := ai.dPmaslo_gaz, StrAIp := protections.dPmaslo_gaz);

  (* Температура газа на выходе нагнетателя *)
  fb_Pmaslo_sm_nizkoe(ai := ai.Pmaslo_sm_nizkoe, StrAIp := protections.Pmaslo_sm_nizkoe);

  (* Температура газа на выходе нагнетателя *)
  fb_Pmaslo_sm_vysokoe(ai := ai.Pmaslo_sm_vysokoe, StrAIp := protections.Pmaslo_sm_vysokoe);

  (* Температура газа на выходе нагнетателя *)
  fb_Vibro_skorost_OPED_T1(ai := ai.Vibro_skorost_OPED_T1, StrAIp := protections.Vibro_skorost_OPED_T1);

  (* Температура газа на выходе нагнетателя *)
  fb_Vibro_skorost_OPED_T2(ai := ai.Vibro_skorost_OYPED_T2, StrAIp := protections.Vibro_skorost_OPED_T2);

  (* Температура газа на выходе нагнетателя *)
  fb_Vibro_skorost_OYP_kolesa_ED_T3(ai := ai.Vibro_skorost_OYP_kolesa_ED_T3, StrAIp := protections.Vibro_skorost_OYP_kolesa_ED_T3);

  (* Температура газа на выходе нагнетателя *)
  fb_Vibro_skorost_OP_kolesa_RH_T4(ai := ai.Vibro_skorost_OP_kolesa_RH_T4, StrAIp := protections.Vibro_skorost_OP_kolesa_RH_T4);

  (* Температура газа на выходе нагнетателя *)
  fb_Vibro_skorost_OP_shesterni_RED_T5(ai := ai.Vibro_skorost_OP_shesterni_RED_T5, StrAIp := protections.Vibro_skorost_OP_shesterni_RED_T5);

  (* Температура газа на выходе нагнетателя *)
  fb_Vibro_skorost_OP_shesterni_RED_T6(ai := ai.Vibro_skorost_OP_shesterni_RED_T6, StrAIp := protections.Vibro_skorost_OP_shesterni_RED_T6);
END_FUNCTION_BLOCK

FUNCTION_BLOCK fb_Kran_Init
  VAR_INPUT
    data_Ini : BOOL;
    ISVALIDREF_statOn : BOOL;
    ISVALIDREF_statOff : BOOL;
    ISVALIDREF_cmdOn : BOOL;
    ISVALIDREF_cmdOff : BOOL;
    ISVALIDREF_inSo : BOOL;
    ISVALIDREF_inSz : BOOL;
    ISVALIDREF_inDp : BOOL          := False;
    continueHoldCommand : TIME;
  END_VAR
  VAR_IN_OUT
    str_Kr : struct_Kran;
  END_VAR
  VAR_OUTPUT
    Init : BOOL          := FALSE;
  END_VAR

  (*****            Функциональный блок переинициализации структуры  Kran          *****)

          Init := False;

      IF data_Ini THEN                            (* Параметрам требуется переинициализация. *)
          str_Kr.ISVALIDREF_statOn                := ISVALIDREF_statOn;
          str_Kr.ISVALIDREF_statOff               := ISVALIDREF_statOff;
          str_Kr.ISVALIDREF_cmdOn                 := ISVALIDREF_cmdOn;
          str_Kr.ISVALIDREF_cmdOff                := ISVALIDREF_cmdOff;
          str_Kr.ISVALIDREF_inSo                  := ISVALIDREF_inSo;
          str_Kr.ISVALIDREF_inSz                  := ISVALIDREF_inSz;
          str_Kr.ISVALIDREF_inDp                  := ISVALIDREF_inDp;
          str_Kr.continueHoldCommand              := continueHoldCommand;

          data_Ini:=False;
          Init := TRUE;
     END_IF;
   IF Init THEN
          ISVALIDREF_statOn:= false;
          ISVALIDREF_statOff:= false;
          ISVALIDREF_cmdOn:= false;
          ISVALIDREF_cmdOff:= false;
          ISVALIDREF_inSo:= false;
          ISVALIDREF_inSz:= false;
          ISVALIDREF_inDp:= false;
          continueHoldCommand:= T#0S;
    END_IF;
END_FUNCTION_BLOCK

FUNCTION_BLOCK fb_Switch_Init
  VAR_INPUT
    data_Ini : BOOL;
    ISVALIDREF_statOn : BOOL;
    ISVALIDREF_statOff : BOOL;
    ISVALIDREF_cmdOn : BOOL;
    ISVALIDREF_cmdOff : BOOL;
    ISVALIDREF_inBreakCmdOn : BOOL;
    ISVALIDREF_inBreakCmdOff : BOOL;
  END_VAR
  VAR_IN_OUT
    str_Sw : struct_Switch;
  END_VAR
  VAR_OUTPUT
    Init : BOOL          := FALSE;
  END_VAR

  (*****            Функциональный блок переинициализации структуры  Switch          *****)

   Init := FALSE;

      IF data_Ini THEN                            (* Параметрам требуется переинициализация. *)
          str_Sw.ISVALIDREF_statOn                := ISVALIDREF_statOn;
          str_Sw.ISVALIDREF_statOff               := ISVALIDREF_statOff;
          str_Sw.ISVALIDREF_cmdOn                 := ISVALIDREF_cmdOn;
          str_Sw.ISVALIDREF_cmdOff                := ISVALIDREF_cmdOff;
          str_Sw.ISVALIDREF_inBreakCmdOn          := ISVALIDREF_inBreakCmdOn;
          str_Sw.ISVALIDREF_inBreakCmdOff         := ISVALIDREF_inBreakCmdOff;
          data_Ini:=FALSE;
          Init := TRUE;
      END_IF;
  IF Init THEN
          ISVALIDREF_statOn:= FALSE;
          ISVALIDREF_statOff:= FALSE;
          ISVALIDREF_cmdOn:= FALSE;
          ISVALIDREF_cmdOff:= FALSE;
          ISVALIDREF_inBreakCmdOn:= FALSE;
          ISVALIDREF_inBreakCmdOff:= FALSE;
  END_IF;
END_FUNCTION_BLOCK

FUNCTION_BLOCK fb_SectionSwitch_Init
  VAR_INPUT
    data_Ini : BOOL;
    ISVALIDREF_statOn : BOOL;
    ISVALIDREF_statOff : BOOL;
    ISVALIDREF_cmdOn : BOOL;
    ISVALIDREF_cmdOff : BOOL;
    ISVALIDREF_inBreakCmdOn : BOOL;
    ISVALIDREF_inBreakCmdOff : BOOL;
    ISVALIDREF_basketRolledIn : BOOL;
    ISVALIDREF_basketRolledOut : BOOL;
    ISVALIDREF_basketTest : BOOL;
  END_VAR
  VAR_IN_OUT
    str_Sw : struct_SectionSwitch;
  END_VAR
  VAR_OUTPUT
    Init : BOOL          := FALSE;
  END_VAR

  (*****            Функциональный блок переинициализации структуры  МВ          *****)

   Init := FALSE;

      IF data_Ini THEN                            (* Параметрам требуется переинициализация. *)
          str_Sw.ISVALIDREF_statOn                := ISVALIDREF_statOn;
          str_Sw.ISVALIDREF_statOff               := ISVALIDREF_statOff;
          str_Sw.ISVALIDREF_cmdOn                 := ISVALIDREF_cmdOn;
          str_Sw.ISVALIDREF_cmdOff                := ISVALIDREF_cmdOff;
          str_Sw.ISVALIDREF_inBreakCmdOn          := ISVALIDREF_inBreakCmdOn;
          str_Sw.ISVALIDREF_inBreakCmdOff         := ISVALIDREF_inBreakCmdOff;
          str_Sw.ISVALIDREF_basketRolledIn        := ISVALIDREF_basketRolledIn;
          str_Sw.ISVALIDREF_basketRolledOut       := ISVALIDREF_basketRolledOut;
          str_Sw.ISVALIDREF_basketTest            := ISVALIDREF_basketTest;
          data_Ini:=FALSE;
          Init := TRUE;
      END_IF;
  IF Init THEN
          ISVALIDREF_statOn:= FALSE;
          ISVALIDREF_statOff:= FALSE;
          ISVALIDREF_cmdOn:= FALSE;
          ISVALIDREF_cmdOff:= FALSE;
          ISVALIDREF_inBreakCmdOn:= FALSE;
          ISVALIDREF_inBreakCmdOff:= FALSE;
          ISVALIDREF_basketRolledIn:= FALSE;
          ISVALIDREF_basketRolledOut:= FALSE;
          ISVALIDREF_basketTest:= FALSE;
  END_IF;
END_FUNCTION_BLOCK

FUNCTION_BLOCK fb_DiscretParametr_Init
  VAR_INPUT
    data_Ini : BOOL;
    currentValue : UINT;
  END_VAR
  VAR_IN_OUT
    strDp : struct_DiscretParametr;
  END_VAR
  VAR_OUTPUT
    Init : BOOL          := FALSE;
  END_VAR

  (*****            Функциональный блок переинициализации дискретного параметра.          *****)

   Init := FALSE;

      IF data_Ini THEN                            (* Параметрам требуется переинициализация. *)
          strDp.currentValue       := currentValue;
          data_Ini:=FALSE;
          Init := TRUE;
      END_IF;
  IF Init THEN
  currentValue:=0;
  END_IF;
END_FUNCTION_BLOCK

FUNCTION_BLOCK fb_singleOutput_Init
  VAR_INPUT
    data_Ini : BOOL;
    inOpcCommandsDisabled : BOOL;
    wait_time : TIME;
  END_VAR
  VAR_IN_OUT
    str_SO : struct_singleOutput;
  END_VAR
  VAR_OUTPUT
    Init : BOOL          := FALSE;
  END_VAR

  (*****            Функциональный блок переинициализации структуры  singleOutput          *****)

  Init := FALSE;

      IF data_Ini THEN                            (* Параметрам требуется переинициализация. *)
          str_SO.inOpcCommandsDisabled    := inOpcCommandsDisabled;
          str_SO.wait_time                := wait_time;

           data_Ini:=FALSE;
          Init := TRUE;
      END_IF;
   IF Init THEN
          inOpcCommandsDisabled := FALSE;
          wait_time := T#0S;
     END_IF;
END_FUNCTION_BLOCK

FUNCTION_BLOCK proc_IM_Init
  VAR_INPUT
    init : BOOL;
  END_VAR
  VAR
    stKr_Ini : fb_Kran_Init;
    stSw_Ini : fb_Switch_Init;
    stOp_Ini : fb_OilPump_Init;
    stSSw_Ini : fb_SectionSwitch_Init;
    stAp_Ini : fb_AnalogParametr_Init;
    stDp_Ini : fb_DiscretParametr_Init;
    stSs_Ini : fb_singleSignal_Init;
    stSo_Ini : fb_singleOutput_Init;
    inits : UINT;
  END_VAR
  VAR_INPUT
    initiales : UINT;
  END_VAR
  VAR_EXTERNAL
    IM : ImConfig;
  END_VAR

  inits := 0; (* Флаг необходимости инициализации структур-дескрипторов *)
                                       (* Стартовая инициализация ИМ *)
  (* Кран 1 *)
  stKr_Ini(data_Ini := true, ISVALIDREF_statOn:=true, ISVALIDREF_statOff:=true,
        ISVALIDREF_cmdOn:=true, ISVALIDREF_cmdOff:=true,
        ISVALIDREF_inSo:=true, ISVALIDREF_inSz:=true,
        str_Kr := IM.Kran1);
  inits := inits + BOOL_TO_UINT(stKr_Ini.Init);

  (* Кран 2 *)
  stKr_Ini(data_Ini := true, ISVALIDREF_statOn:=true, ISVALIDREF_statOff:=true,
        ISVALIDREF_cmdOn:=true, ISVALIDREF_cmdOff:=true,
        ISVALIDREF_inSo:=true, ISVALIDREF_inSz:=true,
        str_Kr := IM.Kran2);
  inits := inits + BOOL_TO_UINT(stKr_Ini.Init);

  (* Кран 3 *)
  stKr_Ini(data_Ini := true, ISVALIDREF_statOn:=true, ISVALIDREF_statOff:=true,
        ISVALIDREF_cmdOn:=true, ISVALIDREF_cmdOff:=true,
        ISVALIDREF_inSo:=true, ISVALIDREF_inSz:=true,
        str_Kr := IM.Kran3);
  inits := inits + BOOL_TO_UINT(stKr_Ini.Init);

  (* Кран 3b *)
  stKr_Ini(data_Ini := true, ISVALIDREF_statOn:=true, ISVALIDREF_statOff:=true,
        ISVALIDREF_cmdOn:=true, ISVALIDREF_cmdOff:=true,
        ISVALIDREF_inSo:=true, ISVALIDREF_inSz:=true,
        str_Kr := IM.Kran3b);
  inits := inits + BOOL_TO_UINT(stKr_Ini.Init);

  (* Кран 4 *)
  stKr_Ini(data_Ini := true, ISVALIDREF_statOn:=true, ISVALIDREF_statOff:=true,
        ISVALIDREF_cmdOn:=true, ISVALIDREF_cmdOff:=true,
        ISVALIDREF_inSo:=true, ISVALIDREF_inSz:=true,
        str_Kr := IM.Kran4);
  inits := inits + BOOL_TO_UINT(stKr_Ini.Init);

  (* Кран 5 *)
  stKr_Ini(data_Ini := true, ISVALIDREF_statOn:=true, ISVALIDREF_statOff:=true,
        ISVALIDREF_cmdOn:=true, ISVALIDREF_cmdOff:=true,
        ISVALIDREF_inSo:=true, ISVALIDREF_inSz:=true, continueHoldCommand:=T#5S,
        str_Kr := IM.Kran5);
  inits := inits + BOOL_TO_UINT(stKr_Ini.Init);

  (* Кран 6 *)
  stKr_Ini(data_Ini := true, ISVALIDREF_statOn:=true, ISVALIDREF_statOff:=true,
        ISVALIDREF_cmdOn:=true, ISVALIDREF_cmdOff:=true,
        str_Kr := IM.Kran6);
  inits := inits + BOOL_TO_UINT(stKr_Ini.Init);

  (* НУ1 Насос уплотнения *)
  stOp_Ini(data_Ini := true, ISVALIDREF_statOn:=true, ISVALIDREF_statOff:=true,
        ISVALIDREF_cmdOn:=true, ISVALIDREF_cmdOff:=true,
        str_Op := IM.nu1);
  inits := inits + BOOL_TO_UINT(stOp_Ini.Init);

  (* НУ2 Насос уплотнения *)
  stOp_Ini(data_Ini := true, ISVALIDREF_statOn:=true, ISVALIDREF_statOff:=true,
        ISVALIDREF_cmdOn:=true, ISVALIDREF_cmdOff:=true,
        str_Op := IM.nu2);
  inits := inits + BOOL_TO_UINT(stOp_Ini.Init);

  (* ПНС Насос смазки *)
  stSw_Ini(data_Ini := true, ISVALIDREF_statOn:=true, ISVALIDREF_statOff:=true,
        ISVALIDREF_cmdOn:=true, ISVALIDREF_cmdOff:=true,
        str_Sw := IM.pns);
  inits := inits + BOOL_TO_UINT(stSw_Ini.Init);

  (* В1 АВОМ вентилятор охлаждения *)
  stSw_Ini(data_Ini := true, ISVALIDREF_statOn:=true, ISVALIDREF_statOff:=true,
        ISVALIDREF_cmdOn:=true, ISVALIDREF_cmdOff:=true,
        str_Sw := IM.v1_Avom);
  inits := inits + BOOL_TO_UINT(stSw_Ini.Init);

  (* В2 АВОМ вентилятор охлаждения *)
  stSw_Ini(data_Ini := true, ISVALIDREF_statOn:=true, ISVALIDREF_statOff:=true,
        ISVALIDREF_cmdOn:=true, ISVALIDREF_cmdOff:=true,
        str_Sw := IM.v2_Avom);
  inits := inits + BOOL_TO_UINT(stSw_Ini.Init);

  (* В3 АВОМ вентилятор охлаждения *)
  stSw_Ini(data_Ini := true, ISVALIDREF_statOn:=true, ISVALIDREF_statOff:=true,
        ISVALIDREF_cmdOn:=true, ISVALIDREF_cmdOff:=true,
        str_Sw := IM.v3_Avom);
  inits := inits + BOOL_TO_UINT(stSw_Ini.Init);

  (* В4 АВОМ вентилятор охлаждения *)
  stSw_Ini(data_Ini := true, ISVALIDREF_statOn:=true, ISVALIDREF_statOff:=true,
        ISVALIDREF_cmdOn:=true, ISVALIDREF_cmdOff:=true,
        str_Sw := IM.v4_Avom);
  inits := inits + BOOL_TO_UINT(stSw_Ini.Init);

  (* МВ масляный выключатель *)
  stSSw_Ini(data_Ini := true, ISVALIDREF_statOn:=true, ISVALIDREF_statOff:=true,
        ISVALIDREF_cmdOn:=true, ISVALIDREF_cmdOff:=true,
        ISVALIDREF_basketRolledIn:=true, ISVALIDREF_basketRolledout:=true,
        str_Sw := IM.mv);
  inits := inits + BOOL_TO_UINT(stSSw_Ini.Init);

  (* В4 АВОМ вентилятор охлаждения *)
  stSw_Ini(data_Ini := true, ISVALIDREF_statOn:=true, ISVALIDREF_statOff:=true,
        ISVALIDREF_cmdOn:=true, ISVALIDREF_cmdOff:=true,
        str_Sw := IM.KaloriferAVOM);
  inits := inits + BOOL_TO_UINT(stSw_Ini.Init);

  (* В4 АВОМ вентилятор охлаждения *)
  stSw_Ini(data_Ini := true, ISVALIDREF_statOn:=true, ISVALIDREF_statOff:=true,
        ISVALIDREF_cmdOn:=true, ISVALIDREF_cmdOff:=true,
        str_Sw := IM.CMN);
  inits := inits + BOOL_TO_UINT(stSw_Ini.Init);

  (* В4 АВОМ вентилятор охлаждения *)
  stSw_Ini(data_Ini := true, ISVALIDREF_statOn:=true, ISVALIDREF_statOff:=true,
        ISVALIDREF_cmdOn:=true, ISVALIDREF_cmdOff:=true,
        str_Sw := IM.TEN_kollectora);
  inits := inits + BOOL_TO_UINT(stSw_Ini.Init);

  (* В4 АВОМ вентилятор охлаждения *)
  stSw_Ini(data_Ini := true, ISVALIDREF_statOn:=true, ISVALIDREF_statOff:=true,
        ISVALIDREF_cmdOn:=true, ISVALIDREF_cmdOff:=true,
        str_Sw := IM.TEN_MB);
  inits := inits + BOOL_TO_UINT(stSw_Ini.Init);

                                       (* Стартовая инициализация singleSignal *)
      (* Перепад давления «газ-газ» на кране 1 ≤1 кгс/см² *)
  stSs_Ini(data_Ini := true, inverse:=FALSE, (*DelayOn:=T#0S, DelayOff:=T#0S,*) str_SS := IM.SingleSignals.dP_maslo_gaz_Less100);
  inits := inits + BOOL_TO_UINT(stSs_Ini.Init);

   (* Осевой сдвиг ротора вправо ≥3,7 кгс/см² *)
  stSs_Ini(data_Ini := true, inverse:=FALSE, (*DelayOn:=T#0S, DelayOff:=T#0S,*) str_SS := IM.SingleSignals.dp_kran1_Less100);
  inits := inits + BOOL_TO_UINT(stSs_Ini.Init);

      (* Пробой вентиля *)
  stSs_Ini(data_Ini := true, inverse:=TRUE, (*DelayOn:=T#0S, DelayOff:=T#0S,*) str_SS := IM.SingleSignals.Vozbud_neispr_tsepey_upr_AVR_pit);
  inits := inits + BOOL_TO_UINT(stSs_Ini.Init);

      (* Работа схемы ресинхронизации *)
  stSs_Ini(data_Ini := true, inverse:=FALSE, (*DelayOn:=T#0S, DelayOff:=T#0S,*) str_SS := IM.SingleSignals.Vozbud_gotovnost);
  inits := inits + BOOL_TO_UINT(stSs_Ini.Init);

      (* Контроль состояния возбудительного устройства  *)
  stSs_Ini(data_Ini := true, inverse:=FALSE, (*DelayOn:=T#0S, DelayOff:=T#0S,*) str_SS := IM.SingleSignals.Vozbud_neispravnost);
  inits := inits + BOOL_TO_UINT(stSs_Ini.Init);

      (* Неисправность форсировки воз-буждения  *)
  stSs_Ini(data_Ini := true, inverse:=FALSE, (*DelayOn:=T#0S, DelayOff:=T#0S,*) str_SS := IM.SingleSignals.SHAVR1_v_rabote);
  inits := inits + BOOL_TO_UINT(stSs_Ini.Init);

    (* Неисправность возбудительного устройства  *)
  stSs_Ini(data_Ini := true, inverse:=FALSE, (*DelayOn:=T#0S, DelayOff:=T#0S,*) str_SS := IM.SingleSignals.SHAVR2_v_rabote);
  inits := inits + BOOL_TO_UINT(stSs_Ini.Init);

    (* Готовность включения БЭО по отказу контроллера  *)
  stSs_Ini(data_Ini := true, inverse:=FALSE, (*DelayOn:=T#0S, DelayOff:=T#0S,*) str_SS := IM.SingleSignals.Avariinoe_otkluch_vikluchatelya);
  inits := inits + BOOL_TO_UINT(stSs_Ini.Init);

    (* Срабатывание БЭАО  *)
  stSs_Ini(data_Ini := true, inverse:=FALSE, (*DelayOn:=T#0S, DelayOff:=T#0S,*) str_SS := IM.SingleSignals.Assinhronnii_hod_peregruzka);
  inits := inits + BOOL_TO_UINT(stSs_Ini.Init);

    (* Выключатель основного ввода питания QF1  в положении включен   *)
  stSs_Ini(data_Ini := true, inverse:=TRUE, (*DelayOn:=T#0S, DelayOff:=T#0S,*) str_SS := IM.SingleSignals.QF1_on);
  inits := inits + BOOL_TO_UINT(stSs_Ini.Init);

    (* Выключатель резервного ввода питания QF2  в положении включен   *)
  stSs_Ini(data_Ini := true, inverse:=TRUE, (*DelayOn:=T#0S, DelayOff:=T#0S,*) str_SS := IM.SingleSignals.QF2_on);
  inits := inits + BOOL_TO_UINT(stSs_Ini.Init);

    (* Выключатель питания кранов:  QF23 110 В в положении включен   *)
  stSs_Ini(data_Ini := true, inverse:=TRUE, (*DelayOn:=T#0S, DelayOff:=T#0S,*) str_SS := IM.SingleSignals.QF23_on);
  inits := inits + BOOL_TO_UINT(stSs_Ini.Init);

    (* Выключатели группы 1: QF4, QF5 в положении включен   *)
  stSs_Ini(data_Ini := true, inverse:=TRUE, (*DelayOn:=T#0S, DelayOff:=T#0S,*) str_SS := IM.SingleSignals.QF4_QF5_on);
  inits := inits + BOOL_TO_UINT(stSs_Ini.Init);

    (* Выключатели группы 2: QF6, QF7 в положении включен   *)
  stSs_Ini(data_Ini := true, inverse:=TRUE, (*DelayOn:=T#0S, DelayOff:=T#0S,*) str_SS := IM.SingleSignals.QF6_QF7_on);
  inits := inits + BOOL_TO_UINT(stSs_Ini.Init);

    (* Выключатели группы 3: QF8, QF9 в положении включен   *)
  stSs_Ini(data_Ini := true, inverse:=TRUE, (*DelayOn:=T#0S, DelayOff:=T#0S,*) str_SS := IM.SingleSignals.QF8_QF9_on);
  inits := inits + BOOL_TO_UINT(stSs_Ini.Init);

    (* Выключатели группы 4: QF10, QF11 в положении включен   *)
  stSs_Ini(data_Ini := true, inverse:=TRUE, (*DelayOn:=T#0S, DelayOff:=T#0S,*) str_SS := IM.SingleSignals.QF10_QF11_on);
  inits := inits + BOOL_TO_UINT(stSs_Ini.Init);

    (* Выключатели группы 5: QF12, QF13 в положении включен   *)
  stSs_Ini(data_Ini := true, inverse:=TRUE, (*DelayOn:=T#0S, DelayOff:=T#0S,*) str_SS := IM.SingleSignals.QF12_QF13_on);
  inits := inits + BOOL_TO_UINT(stSs_Ini.Init);

    (* Выключатели группы 6: QF14, QF15 в положении включен   *)
  stSs_Ini(data_Ini := true, inverse:=TRUE, (*DelayOn:=T#0S, DelayOff:=T#0S,*) str_SS := IM.SingleSignals.QF14_QF15_on);
  inits := inits + BOOL_TO_UINT(stSs_Ini.Init);

    (* Выключатели группы : QF22 в положении включен   *)
  stSs_Ini(data_Ini := true, inverse:=TRUE, (*DelayOn:=T#0S, DelayOff:=T#0S,*) str_SS := IM.SingleSignals.QF22_on);
  inits := inits + BOOL_TO_UINT(stSs_Ini.Init);

    (* Неисправность источников питания группы 1: G1, G2 (=24 В)   *)
  stSs_Ini(data_Ini := true, inverse:=TRUE, (*DelayOn:=T#0S, DelayOff:=T#0S,*) str_SS := IM.SingleSignals.NS_G1_G2);
  inits := inits + BOOL_TO_UINT(stSs_Ini.Init);

    (* Неисправность источников питания группы 2: G3, G4 (=24 В)   *)
  stSs_Ini(data_Ini := true, inverse:=TRUE, (*DelayOn:=T#0S, DelayOff:=T#0S,*) str_SS := IM.SingleSignals.NS_G3_G4);
  inits := inits + BOOL_TO_UINT(stSs_Ini.Init);

    (* Неисправность источников питания внутренних ПТС: G15, G16 (=24 В)   *)
  stSs_Ini(data_Ini := true, inverse:=TRUE, (*DelayOn:=T#0S, DelayOff:=T#0S,*) str_SS := IM.SingleSignals.NS_G15_G16);
  inits := inits + BOOL_TO_UINT(stSs_Ini.Init);

    (* Неисправность источника питания аналоговых сигналов: G17 (=24 В)   *)
  stSs_Ini(data_Ini := true, inverse:=TRUE, (*DelayOn:=T#0S, DelayOff:=T#0S,*) str_SS := IM.SingleSignals.NS_G17);
  inits := inits + BOOL_TO_UINT(stSs_Ini.Init);

    (* Неисправность источников питания группы 3: G5, G6 (=24 В)   *)
  stSs_Ini(data_Ini := true, inverse:=TRUE, (*DelayOn:=T#0S, DelayOff:=T#0S,*) str_SS := IM.SingleSignals.NS_G5_G6);
  inits := inits + BOOL_TO_UINT(stSs_Ini.Init);

    (* Неисправность источников питания группы 4: G7, G8 (=24 В)   *)
  stSs_Ini(data_Ini := true, inverse:=TRUE, (*DelayOn:=T#0S, DelayOff:=T#0S,*) str_SS := IM.SingleSignals.NS_G7_G8);
  inits := inits + BOOL_TO_UINT(stSs_Ini.Init);

    (* Неисправность источников питания внешних цепей: G18, G19 (=24 В)   *)
  stSs_Ini(data_Ini := true, inverse:=TRUE, (*DelayOn:=T#0S, DelayOff:=T#0S,*) str_SS := IM.SingleSignals.NS_G18_G19);
  inits := inits + BOOL_TO_UINT(stSs_Ini.Init);

    (* Неисправность источников питания группы 5: G9, G10, G11, G12 (=110 В)   *)
  stSs_Ini(data_Ini := true, inverse:=TRUE, (*DelayOn:=T#0S, DelayOff:=T#0S,*) str_SS := IM.SingleSignals.NS_G10_G11);
  inits := inits + BOOL_TO_UINT(stSs_Ini.Init);

    (* Неисправность источников питания G13, G14 (=24 В)   *)
  stSs_Ini(data_Ini := true, inverse:=TRUE, (*DelayOn:=T#0S, DelayOff:=T#0S,*) str_SS := IM.SingleSignals.NS_G13_G14);
  inits := inits + BOOL_TO_UINT(stSs_Ini.Init);

      (* Неисправность источников питания G13, G14 (=24 В)   *)
  stSs_Ini(data_Ini := true, inverse:=TRUE, (*DelayOn:=T#0S, DelayOff:=T#0S,*) str_SS := IM.SingleSignals.Uroven_masla_akkum);
  inits := inits + BOOL_TO_UINT(stSs_Ini.Init);

    (* Неисправность источников питания G13, G14 (=24 В)   *)
  stSs_Ini(data_Ini := true, inverse:=TRUE, (*DelayOn:=T#0S, DelayOff:=T#0S,*) str_SS := IM.SingleSignals.BEAO_srabotal);
  inits := inits + BOOL_TO_UINT(stSs_Ini.Init);

    (* Неисправность источников питания G13, G14 (=24 В)   *)
  stSs_Ini(data_Ini := true, inverse:=TRUE, (*DelayOn:=T#0S, DelayOff:=T#0S,*) str_SS := IM.SingleSignals.Chastotny_pusk);
  inits := inits + BOOL_TO_UINT(stSs_Ini.Init);

    (* Неисправность источников питания G13, G14 (=24 В)   *)
  stSs_Ini(data_Ini := true, inverse:=TRUE, (*DelayOn:=T#0S, DelayOff:=T#0S,*) str_SS := IM.SingleSignals.Neuspesh_chastotny_pusk);
  inits := inits + BOOL_TO_UINT(stSs_Ini.Init);

    (* Неисправность источников питания G13, G14 (=24 В)   *)
  stSs_Ini(data_Ini := true, inverse:=TRUE, (*DelayOn:=T#0S, DelayOff:=T#0S,*) str_SS := IM.SingleSignals.Rezhim_ruchnogo_regulirovaniya);
  inits := inits + BOOL_TO_UINT(stSs_Ini.Init);

    (* Неисправность источников питания G13, G14 (=24 В)   *)
  stSs_Ini(data_Ini := true, inverse:=TRUE, (*DelayOn:=T#0S, DelayOff:=T#0S,*) str_SS := IM.SingleSignals.SHU_v_GPA_vkluch);
  inits := inits + BOOL_TO_UINT(stSs_Ini.Init);

    (* Неисправность источников питания G13, G14 (=24 В)   *)
  stSs_Ini(data_Ini := true, inverse:=TRUE, (*DelayOn:=T#0S, DelayOff:=T#0S,*) str_SS := IM.SingleSignals.SHP_v_GPA_vkluch);
  inits := inits + BOOL_TO_UINT(stSs_Ini.Init);

  (* Отключение МВ1 от КНА   *)
  stSs_Ini(data_Ini := true, inverse:=TRUE, (*wait_time:=T#0S,*) str_SS := IM.SingleSignals.NKU1_GPA_on);
  inits := inits + BOOL_TO_UINT(stSs_Ini.Init);

  (* Отключение МВ1 от КНА   *)
  stSs_Ini(data_Ini := true, inverse:=TRUE, (*wait_time:=T#0S,*) str_SS := IM.SingleSignals.NKU2_GPA_on);
  inits := inits + BOOL_TO_UINT(stSs_Ini.Init);

  (* Отключение МВ1 от КНА   *)
  stSs_Ini(data_Ini := true, inverse:=TRUE, (*wait_time:=T#0S,*) str_SS := IM.SingleSignals.AO_KC_ot_SHKS);
  inits := inits + BOOL_TO_UINT(stSs_Ini.Init);

  (* Отключение МВ1 от КНА   *)
  stSs_Ini(data_Ini := true, inverse:=TRUE, (*wait_time:=T#0S,*) str_SS := IM.SingleSignals.AO_GPA_ot_SHU);
  inits := inits + BOOL_TO_UINT(stSs_Ini.Init);

  (* Отключение МВ1 от КНА   *)
  stSs_Ini(data_Ini := true, inverse:=TRUE, (*wait_time:=T#0S,*) str_SS := IM.SingleSignals.Razreshenie_zagruzki_dvig);
  inits := inits + BOOL_TO_UINT(stSs_Ini.Init);

  (* Отключение МВ1 от КНА   *)
  stSs_Ini(data_Ini := true, inverse:=TRUE, (*wait_time:=T#0S,*) str_SS := IM.SingleSignals.Osnovnoy_regul_off);
  inits := inits + BOOL_TO_UINT(stSs_Ini.Init);

  (* Отключение МВ1 от КНА   *)
  stSs_Ini(data_Ini := true, inverse:=TRUE, (*wait_time:=T#0S,*) str_SS := IM.SingleSignals.Voltage_sekcii_norm);
  inits := inits + BOOL_TO_UINT(stSs_Ini.Init);

  (* Отключение МВ1 от КНА   *)
  stSs_Ini(data_Ini := true, inverse:=TRUE, (*wait_time:=T#0S,*) str_SS := IM.SingleSignals.Reactorny_pusk);
  inits := inits + BOOL_TO_UINT(stSs_Ini.Init);

  (* Отключение МВ1 от КНА   *)
  stSs_Ini(data_Ini := true, inverse:=TRUE, (*wait_time:=T#0S,*) str_SS := IM.SingleSignals.NO_GPA_ot_SHU);
  inits := inits + BOOL_TO_UINT(stSs_Ini.Init);

  (* Отключение МВ1 от КНА   *)
  stSs_Ini(data_Ini := true, inverse:=TRUE, (*wait_time:=T#0S,*) str_SS := IM.SingleSignals.AO_GPA_ot_PRU);
  inits := inits + BOOL_TO_UINT(stSs_Ini.Init);

  (* Отключение МВ1 от КНА   *)
  stSs_Ini(data_Ini := true, inverse:=TRUE, (*wait_time:=T#0S,*) str_SS := IM.SingleSignals.Nalichie_BP1);
  inits := inits + BOOL_TO_UINT(stSs_Ini.Init);

  (* Отключение МВ1 от КНА   *)
  stSs_Ini(data_Ini := true, inverse:=TRUE, (*wait_time:=T#0S,*) str_SS := IM.SingleSignals.Nalichie_BP2);
  inits := inits + BOOL_TO_UINT(stSs_Ini.Init);

  (* Отключение МВ1 от КНА   *)
  stSs_Ini(data_Ini := true, inverse:=TRUE, (*wait_time:=T#0S,*) str_SS := IM.SingleSignals.Nalichie_BP3);
  inits := inits + BOOL_TO_UINT(stSs_Ini.Init);

  (* Отключение МВ1 от КНА   *)
  stSs_Ini(data_Ini := true, inverse:=TRUE, (*wait_time:=T#0S,*) str_SS := IM.SingleSignals.Nalichie_BP4);
  inits := inits + BOOL_TO_UINT(stSs_Ini.Init);
